ABB RobotStudio station: Arc_Welding.rsstn

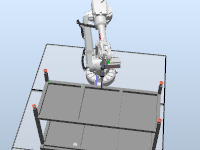
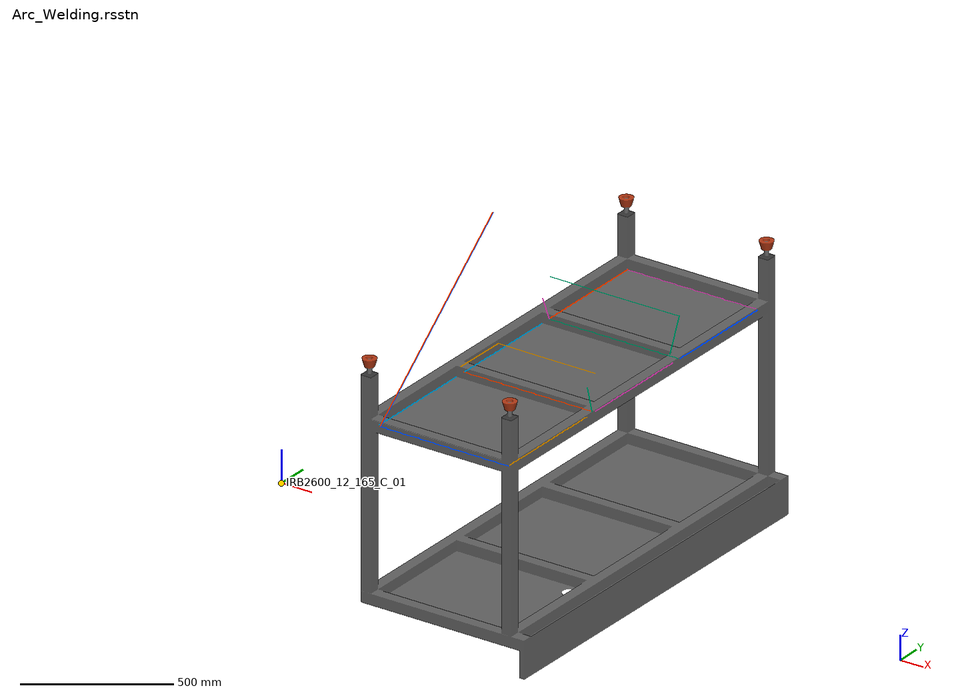
[picture v1: parts stored in the station drawn from their meshes, with robot base, taught points and paths (robot models come from the ABB library and are not in the file)]
Station Arc_Welding (saved by RobotStudio 21.2.9526.0)
Controller Controller_AW
  mechanical unit ROB_1: IRB2600_12_165_C_01, 6 joints, base frame (-416.85, 0, 0) mm
Layout (positions relative to the parent item):
  - IRB2600_12_165_C_01 [mechanism, from Robots\IRB2600_12_165_C_01.rslib] at (-416.85, 0, 0) mm; joint values [0.2384, -0.6663, 0.7884, -0.3764, 0.5482, 0.4666] (rad or m)
  - AW_Gun_PSF_25 [mechanism, from Tools\AW_Gun_PSF_25.rslib] at (157.78, 122.92, 962.92) mm, rotated rx -180 ry 54.2 rz -180 deg
  - Assem1 [graphiccomponentgroup] at (445.82, -642.53, 0) mm, rotated rx 180 ry 0 rz 90 deg
    - Stalas [part] at (21.25, 486.55, -28.09) mm, size 1500 x 650 x 920 mm
    - Part 1 [part] at (22.25, -72.45, -850.09) mm, size 40 x 40 x 35 mm
    - Part 2 [part] at (82.25, -92.45, -879.85) mm, rotated rx 180 ry 0 rz 0 deg, size 51.1 x 51 x 30 mm
    - Hex structural bolt grade C short thread ISO 7412 [part] at (42.25, -92.45, -889.85) mm, rotated rx 180 ry 0 rz 0 deg, size 31.2 x 27 x 80 mm
    - Chamfered plain washer normal ISO 7090 [part] at (42.25, -92.45, -848.59) mm, size 30 x 29.8 x 3 mm
    - Hex flange nut ISO 4161 [part] at (42.25, -92.45, -839.09) mm, size 34.5 x 34.4 x 16 mm
    - Chamfered plain washer normal ISO 7090 [part] at (42.25, 465.55, -848.59) mm, size 30 x 29.8 x 3 mm
    - Hex flange nut ISO 4161 [part] at (42.25, 465.55, -839.09) mm, size 34.5 x 34.4 x 16 mm
    - Hex structural bolt grade C short thread ISO 7412 [part] at (42.25, 465.55, -889.85) mm, rotated rx 180 ry 0 rz 0 deg, size 31.2 x 27 x 80 mm
    - Part 1 [part] at (22.25, 485.55, -850.09) mm, size 40 x 40 x 35 mm
    - Part 2 [part] at (82.25, 465.55, -879.85) mm, rotated rx 180 ry 0 rz 0 deg, size 51.1 x 51 x 30 mm
    - Chamfered plain washer normal ISO 7090 [part] at (1500.25, 465.55, -848.59) mm, size 30 x 29.8 x 3 mm
    - Hex flange nut ISO 4161 [part] at (1500.25, 465.55, -839.09) mm, size 34.5 x 34.4 x 16 mm
    - Hex structural bolt grade C short thread ISO 7412 [part] at (1500.25, 465.55, -889.85) mm, rotated rx 180 ry 0 rz 0 deg, size 31.2 x 27 x 80 mm
    - Part 1 [part] at (1480.25, 485.55, -850.09) mm, size 40 x 40 x 35 mm
    - Part 2 [part] at (1540.25, 465.55, -879.85) mm, rotated rx 180 ry 0 rz 0 deg, size 51.1 x 51 x 30 mm
    - Chamfered plain washer normal ISO 7090 [part] at (1500.25, -92.45, -848.59) mm, size 30 x 29.8 x 3 mm
    - Hex flange nut ISO 4161 [part] at (1500.25, -92.45, -839.09) mm, size 34.5 x 34.4 x 16 mm
    - Hex structural bolt grade C short thread ISO 7412 [part] at (1500.25, -92.45, -889.85) mm, rotated rx 180 ry 0 rz 0 deg, size 31.2 x 27 x 80 mm
    - Part 1 [part] at (1480.25, -72.45, -850.09) mm, size 40 x 40 x 35 mm
    - Part 2 [part] at (1540.25, -92.45, -879.85) mm, rotated rx 180 ry 0 rz 0 deg, size 51.1 x 51 x 30 mm
    - Part 1 [part] at (62.25, 445.55, -28.09) mm, size 1418 x 598 x 40 mm
    - Part 1 [part] at (62.25, 445.55, -660.09) mm, size 1418 x 598 x 40 mm
    - Part 1 [part] at (64.25, 445.55, -660.09) mm, rotated rx 0 ry 90 rz 0 deg, size 40 x 519 x 40 mm
    - Part 1 [part] at (1478.25, 446.55, -660.09) mm, size 40 x 519 x 40 mm
    - Part 1 [part] at (1480.25, 445.55, -28.09) mm, size 40 x 519 x 40 mm
    - Part 1 [part] at (22.25, 445.55, -28.09) mm, size 40 x 519 x 40 mm
Attachment: AW_Gun_PSF_25 is attached to IRB2600_12_165_C_01 / Link6
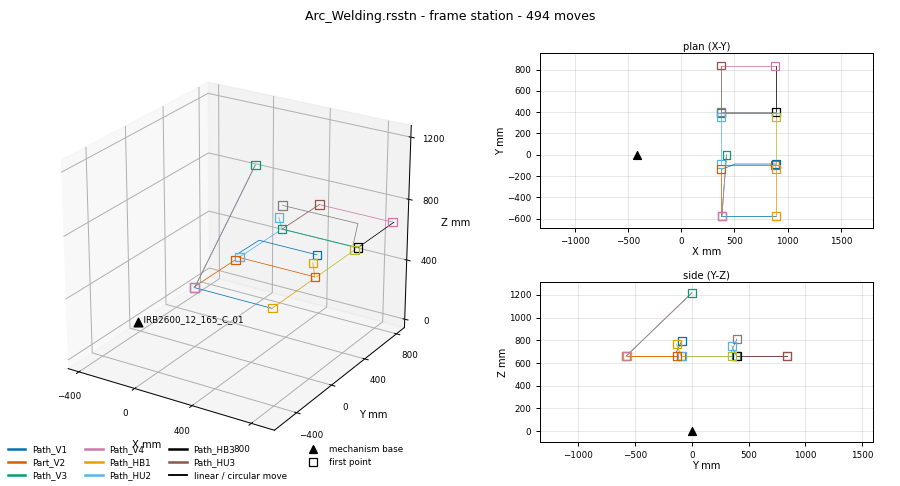
[picture p0: tool path of Arc_Welding.rsstn in frame station, 494 of 494 moves have a stored position in this frame; points joined in program order, loops and branches not executed]
Targets, tools, work objects and paths stored in the station, written as RAPID:
! task T_ROB1
MODULE CalibData
  PERS tooldata AW_Gun:=[TRUE,[[119.5,0,352],[0.890213743,0,0.455543074,0]],[1,[0,0,100],[1,0,0,0],0,0,0]];
ENDMODULE

! task T_ROB1
MODULE Module1
  CONST robtarget Target_10:=[[891.374984158,-578.28436321,660.090342283],[0,0,1,0],[0,0,0,0],[9E+09,9E+09,9E+09,9E+09,9E+09,9E+09]];
  CONST robtarget Target_20:=[[881.374984158,-578.28436321,660.090342283],[0,0,1,0],[0,0,0,0],[9E+09,9E+09,9E+09,9E+09,9E+09,9E+09]];
  CONST robtarget Target_30:=[[871.374984158,-578.28436321,660.090342283],[0,0,1,0],[0,0,0,0],[9E+09,9E+09,9E+09,9E+09,9E+09,9E+09]];
  CONST robtarget Target_40:=[[861.374984158,-578.28436321,660.090342283],[0,0,1,0],[0,0,0,0],[9E+09,9E+09,9E+09,9E+09,9E+09,9E+09]];
  CONST robtarget Target_50:=[[851.374984158,-578.28436321,660.090342283],[0,0,1,0],[0,0,0,0],[9E+09,9E+09,9E+09,9E+09,9E+09,9E+09]];
  CONST robtarget Target_60:=[[841.374984158,-578.28436321,660.090342283],[0,0,1,0],[0,0,0,0],[9E+09,9E+09,9E+09,9E+09,9E+09,9E+09]];
  CONST robtarget Target_70:=[[831.374984158,-578.28436321,660.090342283],[0,0,1,0],[0,0,0,0],[9E+09,9E+09,9E+09,9E+09,9E+09,9E+09]];
  CONST robtarget Target_80:=[[821.374984158,-578.28436321,660.090342283],[0,0,1,0],[0,0,0,0],[9E+09,9E+09,9E+09,9E+09,9E+09,9E+09]];
  CONST robtarget Target_90:=[[811.374984158,-578.28436321,660.090342283],[0,0,1,0],[0,0,0,0],[9E+09,9E+09,9E+09,9E+09,9E+09,9E+09]];
  CONST robtarget Target_100:=[[801.374984158,-578.28436321,660.090342283],[0,0,1,0],[0,0,0,0],[9E+09,9E+09,9E+09,9E+09,9E+09,9E+09]];
  CONST robtarget Target_110:=[[791.374984158,-578.28436321,660.090342283],[0,0,1,0],[0,0,0,0],[9E+09,9E+09,9E+09,9E+09,9E+09,9E+09]];
  CONST robtarget Target_120:=[[781.374984158,-578.28436321,660.090342283],[0,0,1,0],[0,0,0,0],[9E+09,9E+09,9E+09,9E+09,9E+09,9E+09]];
  CONST robtarget Target_130:=[[771.374984158,-578.28436321,660.090342283],[0,0,1,0],[0,0,0,0],[9E+09,9E+09,9E+09,9E+09,9E+09,9E+09]];
  CONST robtarget Target_140:=[[761.374984158,-578.28436321,660.090342283],[0,0,1,0],[0,0,0,0],[9E+09,9E+09,9E+09,9E+09,9E+09,9E+09]];
  CONST robtarget Target_150:=[[751.374984158,-578.28436321,660.090342283],[0,0,1,0],[0,0,0,0],[9E+09,9E+09,9E+09,9E+09,9E+09,9E+09]];
  CONST robtarget Target_160:=[[741.374984158,-578.28436321,660.090342283],[0,0,1,0],[0,0,0,0],[9E+09,9E+09,9E+09,9E+09,9E+09,9E+09]];
  CONST robtarget Target_170:=[[731.374984158,-578.28436321,660.090342283],[0,0,1,0],[0,0,0,0],[9E+09,9E+09,9E+09,9E+09,9E+09,9E+09]];
  CONST robtarget Target_180:=[[721.374984158,-578.28436321,660.090342283],[0,0,1,0],[0,0,0,0],[9E+09,9E+09,9E+09,9E+09,9E+09,9E+09]];
  CONST robtarget Target_190:=[[711.374984158,-578.28436321,660.090342283],[0,0,1,0],[0,0,0,0],[9E+09,9E+09,9E+09,9E+09,9E+09,9E+09]];
  CONST robtarget Target_200:=[[701.374984158,-578.28436321,660.090342283],[0,0,1,0],[0,0,0,0],[9E+09,9E+09,9E+09,9E+09,9E+09,9E+09]];
  CONST robtarget Target_210:=[[691.374984158,-578.28436321,660.090342283],[0,0,1,0],[0,0,0,0],[9E+09,9E+09,9E+09,9E+09,9E+09,9E+09]];
  CONST robtarget Target_220:=[[681.374984158,-578.28436321,660.090342283],[0,0,1,0],[0,0,0,0],[9E+09,9E+09,9E+09,9E+09,9E+09,9E+09]];
  CONST robtarget Target_230:=[[671.374984158,-578.28436321,660.090342283],[0,0,1,0],[0,0,0,0],[9E+09,9E+09,9E+09,9E+09,9E+09,9E+09]];
  CONST robtarget Target_240:=[[661.374984158,-578.28436321,660.090342283],[0,0,1,0],[0,0,0,0],[9E+09,9E+09,9E+09,9E+09,9E+09,9E+09]];
  CONST robtarget Target_250:=[[651.374984158,-578.28436321,660.090342283],[0,0,1,0],[0,0,0,0],[9E+09,9E+09,9E+09,9E+09,9E+09,9E+09]];
  CONST robtarget Target_260:=[[641.374984158,-578.28436321,660.090342283],[0,0,1,0],[0,0,0,0],[9E+09,9E+09,9E+09,9E+09,9E+09,9E+09]];
  CONST robtarget Target_270:=[[631.374984158,-578.28436321,660.090342283],[0,0,1,0],[0,0,0,0],[9E+09,9E+09,9E+09,9E+09,9E+09,9E+09]];
  CONST robtarget Target_280:=[[621.374984158,-578.28436321,660.090342283],[0,0,1,0],[0,0,0,0],[9E+09,9E+09,9E+09,9E+09,9E+09,9E+09]];
  CONST robtarget Target_290:=[[611.374984158,-578.28436321,660.090342283],[0,0,1,0],[0,0,0,0],[9E+09,9E+09,9E+09,9E+09,9E+09,9E+09]];
  CONST robtarget Target_300:=[[601.374984158,-578.28436321,660.090342283],[0,0,1,0],[0,0,0,0],[9E+09,9E+09,9E+09,9E+09,9E+09,9E+09]];
  CONST robtarget Target_310:=[[591.374984158,-578.28436321,660.090342283],[0,0,1,0],[0,0,0,0],[9E+09,9E+09,9E+09,9E+09,9E+09,9E+09]];
  CONST robtarget Target_320:=[[581.374984158,-578.28436321,660.090342283],[0,0,1,0],[0,0,0,0],[9E+09,9E+09,9E+09,9E+09,9E+09,9E+09]];
  CONST robtarget Target_330:=[[571.374984158,-578.28436321,660.090342283],[0,0,1,0],[0,0,0,0],[9E+09,9E+09,9E+09,9E+09,9E+09,9E+09]];
  CONST robtarget Target_340:=[[561.374984158,-578.28436321,660.090342283],[0,0,1,0],[0,0,0,0],[9E+09,9E+09,9E+09,9E+09,9E+09,9E+09]];
  CONST robtarget Target_350:=[[551.374984158,-578.28436321,660.090342283],[0,0,1,0],[0,0,0,0],[9E+09,9E+09,9E+09,9E+09,9E+09,9E+09]];
  CONST robtarget Target_360:=[[541.374984158,-578.28436321,660.090342283],[0,0,1,0],[0,0,0,0],[9E+09,9E+09,9E+09,9E+09,9E+09,9E+09]];
  CONST robtarget Target_370:=[[531.374984158,-578.28436321,660.090342283],[0,0,1,0],[0,0,0,0],[9E+09,9E+09,9E+09,9E+09,9E+09,9E+09]];
  CONST robtarget Target_380:=[[521.374984158,-578.28436321,660.090342283],[0,0,1,0],[0,0,0,0],[9E+09,9E+09,9E+09,9E+09,9E+09,9E+09]];
  CONST robtarget Target_390:=[[511.374984158,-578.28436321,660.090342283],[0,0,1,0],[0,0,0,0],[9E+09,9E+09,9E+09,9E+09,9E+09,9E+09]];
  CONST robtarget Target_400:=[[501.374984158,-578.28436321,660.090342283],[0,0,1,0],[0,0,0,0],[9E+09,9E+09,9E+09,9E+09,9E+09,9E+09]];
  CONST robtarget Target_410:=[[491.374984158,-578.28436321,660.090342283],[0,0,1,0],[0,0,0,0],[9E+09,9E+09,9E+09,9E+09,9E+09,9E+09]];
  CONST robtarget Target_420:=[[481.374984158,-578.28436321,660.090342283],[0,0,1,0],[0,0,0,0],[9E+09,9E+09,9E+09,9E+09,9E+09,9E+09]];
  CONST robtarget Target_430:=[[471.374984158,-578.28436321,660.090342283],[0,0,1,0],[0,0,0,0],[9E+09,9E+09,9E+09,9E+09,9E+09,9E+09]];
  CONST robtarget Target_440:=[[461.374984158,-578.28436321,660.090342283],[0,0,1,0],[0,0,0,0],[9E+09,9E+09,9E+09,9E+09,9E+09,9E+09]];
  CONST robtarget Target_450:=[[451.374984158,-578.28436321,660.090342283],[0,0,1,0],[0,0,0,0],[9E+09,9E+09,9E+09,9E+09,9E+09,9E+09]];
  CONST robtarget Target_460:=[[441.374984158,-578.28436321,660.090342283],[0,0,1,0],[0,0,0,0],[9E+09,9E+09,9E+09,9E+09,9E+09,9E+09]];
  CONST robtarget Target_470:=[[431.374984158,-578.28436321,660.090342283],[0,0,1,0],[0,0,0,0],[9E+09,9E+09,9E+09,9E+09,9E+09,9E+09]];
  CONST robtarget Target_480:=[[421.374984158,-578.28436321,660.090342283],[0,0,1,0],[0,0,0,0],[9E+09,9E+09,9E+09,9E+09,9E+09,9E+09]];
  CONST robtarget Target_490:=[[411.374984158,-578.28436321,660.090342283],[0,0,1,0],[0,0,0,0],[9E+09,9E+09,9E+09,9E+09,9E+09,9E+09]];
  CONST robtarget Target_500:=[[401.374984158,-578.28436321,660.090342283],[0,0,1,0],[0,0,0,0],[9E+09,9E+09,9E+09,9E+09,9E+09,9E+09]];
  CONST robtarget Target_510:=[[391.374984158,-578.28436321,660.090342283],[0,0,1,0],[0,0,0,0],[9E+09,9E+09,9E+09,9E+09,9E+09,9E+09]];
  CONST robtarget Target_520:=[[381.374984158,-578.28436321,660.090342283],[0,0,1,0],[0,0,0,0],[9E+09,9E+09,9E+09,9E+09,9E+09,9E+09]];
  CONST robtarget Target_530:=[[373.374984158,-133.68436321,660.090342283],[0.5,0.5,-0.5,-0.5],[0,0,0,0],[9E+09,9E+09,9E+09,9E+09,9E+09,9E+09]];
  CONST robtarget Target_540:=[[373.374984158,-580.28436321,660.090342283],[0.5,0.5,-0.5,-0.5],[0,0,0,0],[9E+09,9E+09,9E+09,9E+09,9E+09,9E+09]];
  CONST robtarget Target_570:=[[373.374984158,-93.68436321,660.090342283],[0,0,1,0],[0,0,0,0],[9E+09,9E+09,9E+09,9E+09,9E+09,9E+09]];
  CONST robtarget Target_580:=[[383.374984158,-93.68436321,660.090342283],[0,0,1,0],[0,0,0,0],[9E+09,9E+09,9E+09,9E+09,9E+09,9E+09]];
  CONST robtarget Target_590:=[[393.374984158,-93.68436321,660.090342283],[0,0,1,0],[0,0,0,0],[9E+09,9E+09,9E+09,9E+09,9E+09,9E+09]];
  CONST robtarget Target_600:=[[403.374984158,-93.68436321,660.090342283],[0,0,1,0],[0,0,0,0],[9E+09,9E+09,9E+09,9E+09,9E+09,9E+09]];
  CONST robtarget Target_610:=[[413.374984158,-93.68436321,660.090342283],[0,0,1,0],[0,0,0,0],[9E+09,9E+09,9E+09,9E+09,9E+09,9E+09]];
  CONST robtarget Target_620:=[[423.374984158,-93.68436321,660.090342283],[0,0,1,0],[0,0,0,0],[9E+09,9E+09,9E+09,9E+09,9E+09,9E+09]];
  CONST robtarget Target_630:=[[433.374984158,-93.68436321,660.090342283],[0,0,1,0],[0,0,0,0],[9E+09,9E+09,9E+09,9E+09,9E+09,9E+09]];
  CONST robtarget Target_640:=[[443.374984158,-93.68436321,660.090342283],[0,0,1,0],[0,0,0,0],[9E+09,9E+09,9E+09,9E+09,9E+09,9E+09]];
  CONST robtarget Target_650:=[[453.374984158,-93.68436321,660.090342283],[0,0,1,0],[0,0,0,0],[9E+09,9E+09,9E+09,9E+09,9E+09,9E+09]];
  CONST robtarget Target_660:=[[463.374984158,-93.68436321,660.090342283],[0,0,1,0],[0,0,0,0],[9E+09,9E+09,9E+09,9E+09,9E+09,9E+09]];
  CONST robtarget Target_670:=[[473.374984158,-93.68436321,660.090342283],[0,0,1,0],[0,0,0,0],[9E+09,9E+09,9E+09,9E+09,9E+09,9E+09]];
  CONST robtarget Target_680:=[[483.374984158,-93.68436321,660.090342283],[0,0,1,0],[0,0,0,0],[9E+09,9E+09,9E+09,9E+09,9E+09,9E+09]];
  CONST robtarget Target_690:=[[493.374984158,-93.68436321,660.090342283],[0,0,1,0],[0,0,0,0],[9E+09,9E+09,9E+09,9E+09,9E+09,9E+09]];
  CONST robtarget Target_700:=[[503.374984158,-93.68436321,660.090342283],[0,0,1,0],[0,0,0,0],[9E+09,9E+09,9E+09,9E+09,9E+09,9E+09]];
  CONST robtarget Target_710:=[[513.374984158,-93.68436321,660.090342283],[0,0,1,0],[0,0,0,0],[9E+09,9E+09,9E+09,9E+09,9E+09,9E+09]];
  CONST robtarget Target_720:=[[523.374984158,-93.68436321,660.090342283],[0,0,1,0],[0,0,0,0],[9E+09,9E+09,9E+09,9E+09,9E+09,9E+09]];
  CONST robtarget Target_730:=[[533.374984158,-93.68436321,660.090342283],[0,0,1,0],[0,0,0,0],[9E+09,9E+09,9E+09,9E+09,9E+09,9E+09]];
  CONST robtarget Target_740:=[[543.374984158,-93.68436321,660.090342283],[0,0,1,0],[0,0,0,0],[9E+09,9E+09,9E+09,9E+09,9E+09,9E+09]];
  CONST robtarget Target_750:=[[553.374984158,-93.68436321,660.090342283],[0,0,1,0],[0,0,0,0],[9E+09,9E+09,9E+09,9E+09,9E+09,9E+09]];
  CONST robtarget Target_760:=[[563.374984158,-93.68436321,660.090342283],[0,0,1,0],[0,0,0,0],[9E+09,9E+09,9E+09,9E+09,9E+09,9E+09]];
  CONST robtarget Target_770:=[[573.374984158,-93.68436321,660.090342283],[0,0,1,0],[0,0,0,0],[9E+09,9E+09,9E+09,9E+09,9E+09,9E+09]];
  CONST robtarget Target_780:=[[583.374984158,-93.68436321,660.090342283],[0,0,1,0],[0,0,0,0],[9E+09,9E+09,9E+09,9E+09,9E+09,9E+09]];
  CONST robtarget Target_790:=[[593.374984158,-93.68436321,660.090342283],[0,0,1,0],[0,0,0,0],[9E+09,9E+09,9E+09,9E+09,9E+09,9E+09]];
  CONST robtarget Target_800:=[[603.374984158,-93.68436321,660.090342283],[0,0,1,0],[0,0,0,0],[9E+09,9E+09,9E+09,9E+09,9E+09,9E+09]];
  CONST robtarget Target_810:=[[613.374984158,-93.68436321,660.090342283],[0,0,1,0],[0,0,0,0],[9E+09,9E+09,9E+09,9E+09,9E+09,9E+09]];
  CONST robtarget Target_820:=[[623.374984158,-93.68436321,660.090342283],[0,0,1,0],[0,0,0,0],[9E+09,9E+09,9E+09,9E+09,9E+09,9E+09]];
  CONST robtarget Target_830:=[[633.374984158,-93.68436321,660.090342283],[0,0,1,0],[0,0,0,0],[9E+09,9E+09,9E+09,9E+09,9E+09,9E+09]];
  CONST robtarget Target_840:=[[643.374984158,-93.68436321,660.090342283],[0,0,1,0],[0,0,0,0],[9E+09,9E+09,9E+09,9E+09,9E+09,9E+09]];
  CONST robtarget Target_850:=[[653.374984158,-93.68436321,660.090342283],[0,0,1,0],[0,0,0,0],[9E+09,9E+09,9E+09,9E+09,9E+09,9E+09]];
  CONST robtarget Target_860:=[[663.374984158,-93.68436321,660.090342283],[0,0,1,0],[0,0,0,0],[9E+09,9E+09,9E+09,9E+09,9E+09,9E+09]];
  CONST robtarget Target_870:=[[673.374984158,-93.68436321,660.090342283],[0,0,1,0],[0,0,0,0],[9E+09,9E+09,9E+09,9E+09,9E+09,9E+09]];
  CONST robtarget Target_880:=[[683.374984158,-93.68436321,660.090342283],[0,0,1,0],[0,0,0,0],[9E+09,9E+09,9E+09,9E+09,9E+09,9E+09]];
  CONST robtarget Target_890:=[[693.374984158,-93.68436321,660.090342283],[0,0,1,0],[0,0,0,0],[9E+09,9E+09,9E+09,9E+09,9E+09,9E+09]];
  CONST robtarget Target_900:=[[703.374984158,-93.68436321,660.090342283],[0,0,1,0],[0,0,0,0],[9E+09,9E+09,9E+09,9E+09,9E+09,9E+09]];
  CONST robtarget Target_910:=[[713.374984158,-93.68436321,660.090342283],[0,0,1,0],[0,0,0,0],[9E+09,9E+09,9E+09,9E+09,9E+09,9E+09]];
  CONST robtarget Target_920:=[[723.374984158,-93.68436321,660.090342283],[0,0,1,0],[0,0,0,0],[9E+09,9E+09,9E+09,9E+09,9E+09,9E+09]];
  CONST robtarget Target_930:=[[733.374984158,-93.68436321,660.090342283],[0,0,1,0],[0,0,0,0],[9E+09,9E+09,9E+09,9E+09,9E+09,9E+09]];
  CONST robtarget Target_940:=[[743.374984158,-93.68436321,660.090342283],[0,0,1,0],[0,0,0,0],[9E+09,9E+09,9E+09,9E+09,9E+09,9E+09]];
  CONST robtarget Target_950:=[[753.374984158,-93.68436321,660.090342283],[0,0,1,0],[0,0,0,0],[9E+09,9E+09,9E+09,9E+09,9E+09,9E+09]];
  CONST robtarget Target_960:=[[763.374984158,-93.68436321,660.090342283],[0,0,1,0],[0,0,0,0],[9E+09,9E+09,9E+09,9E+09,9E+09,9E+09]];
  CONST robtarget Target_970:=[[773.374984158,-93.68436321,660.090342283],[0,0,1,0],[0,0,0,0],[9E+09,9E+09,9E+09,9E+09,9E+09,9E+09]];
  CONST robtarget Target_980:=[[783.374984158,-93.68436321,660.090342283],[0,0,1,0],[0,0,0,0],[9E+09,9E+09,9E+09,9E+09,9E+09,9E+09]];
  CONST robtarget Target_990:=[[793.374984158,-93.68436321,660.090342283],[0,0,1,0],[0,0,0,0],[9E+09,9E+09,9E+09,9E+09,9E+09,9E+09]];
  CONST robtarget Target_1000:=[[803.374984158,-93.68436321,660.090342283],[0,0,1,0],[0,0,0,0],[9E+09,9E+09,9E+09,9E+09,9E+09,9E+09]];
  CONST robtarget Target_1010:=[[813.374984158,-93.68436321,660.090342283],[0,0,1,0],[0,0,0,0],[9E+09,9E+09,9E+09,9E+09,9E+09,9E+09]];
  CONST robtarget Target_1020:=[[823.374984158,-93.68436321,660.090342283],[0,0,1,0],[0,0,0,0],[9E+09,9E+09,9E+09,9E+09,9E+09,9E+09]];
  CONST robtarget Target_1030:=[[833.374984158,-93.68436321,660.090342283],[0,0,1,0],[0,0,0,0],[9E+09,9E+09,9E+09,9E+09,9E+09,9E+09]];
  CONST robtarget Target_1040:=[[843.374984158,-93.68436321,660.090342283],[0,0,1,0],[0,0,0,0],[9E+09,9E+09,9E+09,9E+09,9E+09,9E+09]];
  CONST robtarget Target_1050:=[[853.374984158,-93.68436321,660.090342283],[0,0,1,0],[0,0,0,0],[9E+09,9E+09,9E+09,9E+09,9E+09,9E+09]];
  CONST robtarget Target_1060:=[[863.374984158,-93.68436321,660.090342283],[0,0,1,0],[0,0,0,0],[9E+09,9E+09,9E+09,9E+09,9E+09,9E+09]];
  CONST robtarget Target_1070:=[[873.374984158,-93.68436321,660.090342283],[0,0,1,0],[0,0,0,0],[9E+09,9E+09,9E+09,9E+09,9E+09,9E+09]];
  CONST robtarget Target_1080:=[[883.374984158,-93.68436321,660.090342283],[0,0,1,0],[0,0,0,0],[9E+09,9E+09,9E+09,9E+09,9E+09,9E+09]];
  CONST robtarget Target_1090:=[[373.374984158,392.91563679,660.090342283],[0,0,1,0],[0,0,0,0],[9E+09,9E+09,9E+09,9E+09,9E+09,9E+09]];
  CONST robtarget Target_1100:=[[383.374984158,392.91563679,660.090342283],[0,0,1,0],[0,0,0,0],[9E+09,9E+09,9E+09,9E+09,9E+09,9E+09]];
  CONST robtarget Target_1110:=[[393.374984158,392.91563679,660.090342283],[0,0,1,0],[0,0,0,0],[9E+09,9E+09,9E+09,9E+09,9E+09,9E+09]];
  CONST robtarget Target_1120:=[[403.374984158,392.91563679,660.090342283],[0,0,1,0],[0,0,0,0],[9E+09,9E+09,9E+09,9E+09,9E+09,9E+09]];
  CONST robtarget Target_1130:=[[413.374984158,392.91563679,660.090342283],[0,0,1,0],[0,0,0,0],[9E+09,9E+09,9E+09,9E+09,9E+09,9E+09]];
  CONST robtarget Target_1140:=[[423.374984158,392.91563679,660.090342283],[0,0,1,0],[0,0,0,0],[9E+09,9E+09,9E+09,9E+09,9E+09,9E+09]];
  CONST robtarget Target_1150:=[[433.374984158,392.91563679,660.090342283],[0,0,1,0],[0,0,0,0],[9E+09,9E+09,9E+09,9E+09,9E+09,9E+09]];
  CONST robtarget Target_1160:=[[443.374984158,392.91563679,660.090342283],[0,0,1,0],[0,0,0,0],[9E+09,9E+09,9E+09,9E+09,9E+09,9E+09]];
  CONST robtarget Target_1170:=[[453.374984158,392.91563679,660.090342283],[0,0,1,0],[0,0,0,0],[9E+09,9E+09,9E+09,9E+09,9E+09,9E+09]];
  CONST robtarget Target_1180:=[[463.374984158,392.91563679,660.090342283],[0,0,1,0],[0,0,0,0],[9E+09,9E+09,9E+09,9E+09,9E+09,9E+09]];
  CONST robtarget Target_1190:=[[473.374984158,392.91563679,660.090342283],[0,0,1,0],[0,0,0,0],[9E+09,9E+09,9E+09,9E+09,9E+09,9E+09]];
  CONST robtarget Target_1200:=[[483.374984158,392.91563679,660.090342283],[0,0,1,0],[0,0,0,0],[9E+09,9E+09,9E+09,9E+09,9E+09,9E+09]];
  CONST robtarget Target_1210:=[[493.374984158,392.91563679,660.090342283],[0,0,1,0],[0,0,0,0],[9E+09,9E+09,9E+09,9E+09,9E+09,9E+09]];
  CONST robtarget Target_1220:=[[503.374984158,392.91563679,660.090342283],[0,0,1,0],[0,0,0,0],[9E+09,9E+09,9E+09,9E+09,9E+09,9E+09]];
  CONST robtarget Target_1230:=[[513.374984158,392.91563679,660.090342283],[0,0,1,0],[0,0,0,0],[9E+09,9E+09,9E+09,9E+09,9E+09,9E+09]];
  CONST robtarget Target_1240:=[[523.374984158,392.91563679,660.090342283],[0,0,1,0],[0,0,0,0],[9E+09,9E+09,9E+09,9E+09,9E+09,9E+09]];
  CONST robtarget Target_1250:=[[533.374984158,392.91563679,660.090342283],[0,0,1,0],[0,0,0,0],[9E+09,9E+09,9E+09,9E+09,9E+09,9E+09]];
  CONST robtarget Target_1260:=[[543.374984158,392.91563679,660.090342283],[0,0,1,0],[0,0,0,0],[9E+09,9E+09,9E+09,9E+09,9E+09,9E+09]];
  CONST robtarget Target_1270:=[[553.374984158,392.91563679,660.090342283],[0,0,1,0],[0,0,0,0],[9E+09,9E+09,9E+09,9E+09,9E+09,9E+09]];
  CONST robtarget Target_1280:=[[563.374984158,392.91563679,660.090342283],[0,0,1,0],[0,0,0,0],[9E+09,9E+09,9E+09,9E+09,9E+09,9E+09]];
  CONST robtarget Target_1290:=[[573.374984158,392.91563679,660.090342283],[0,0,1,0],[0,0,0,0],[9E+09,9E+09,9E+09,9E+09,9E+09,9E+09]];
  CONST robtarget Target_1300:=[[583.374984158,392.91563679,660.090342283],[0,0,1,0],[0,0,0,0],[9E+09,9E+09,9E+09,9E+09,9E+09,9E+09]];
  CONST robtarget Target_1310:=[[593.374984158,392.91563679,660.090342283],[0,0,1,0],[0,0,0,0],[9E+09,9E+09,9E+09,9E+09,9E+09,9E+09]];
  CONST robtarget Target_1320:=[[603.374984158,392.91563679,660.090342283],[0,0,1,0],[0,0,0,0],[9E+09,9E+09,9E+09,9E+09,9E+09,9E+09]];
  CONST robtarget Target_1330:=[[613.374984158,392.91563679,660.090342283],[0,0,1,0],[0,0,0,0],[9E+09,9E+09,9E+09,9E+09,9E+09,9E+09]];
  CONST robtarget Target_1340:=[[623.374984158,392.91563679,660.090342283],[0,0,1,0],[0,0,0,0],[9E+09,9E+09,9E+09,9E+09,9E+09,9E+09]];
  CONST robtarget Target_1350:=[[633.374984158,392.91563679,660.090342283],[0,0,1,0],[0,0,0,0],[9E+09,9E+09,9E+09,9E+09,9E+09,9E+09]];
  CONST robtarget Target_1360:=[[643.374984158,392.91563679,660.090342283],[0,0,1,0],[0,0,0,0],[9E+09,9E+09,9E+09,9E+09,9E+09,9E+09]];
  CONST robtarget Target_1370:=[[653.374984158,392.91563679,660.090342283],[0,0,1,0],[0,0,0,0],[9E+09,9E+09,9E+09,9E+09,9E+09,9E+09]];
  CONST robtarget Target_1380:=[[663.374984158,392.91563679,660.090342283],[0,0,1,0],[0,0,0,0],[9E+09,9E+09,9E+09,9E+09,9E+09,9E+09]];
  CONST robtarget Target_1390:=[[673.374984158,392.91563679,660.090342283],[0,0,1,0],[0,0,0,0],[9E+09,9E+09,9E+09,9E+09,9E+09,9E+09]];
  CONST robtarget Target_1400:=[[683.374984158,392.91563679,660.090342283],[0,0,1,0],[0,0,0,0],[9E+09,9E+09,9E+09,9E+09,9E+09,9E+09]];
  CONST robtarget Target_1410:=[[693.374984158,392.91563679,660.090342283],[0,0,1,0],[0,0,0,0],[9E+09,9E+09,9E+09,9E+09,9E+09,9E+09]];
  CONST robtarget Target_1420:=[[703.374984158,392.91563679,660.090342283],[0,0,1,0],[0,0,0,0],[9E+09,9E+09,9E+09,9E+09,9E+09,9E+09]];
  CONST robtarget Target_1430:=[[713.374984158,392.91563679,660.090342283],[0,0,1,0],[0,0,0,0],[9E+09,9E+09,9E+09,9E+09,9E+09,9E+09]];
  CONST robtarget Target_1440:=[[723.374984158,392.91563679,660.090342283],[0,0,1,0],[0,0,0,0],[9E+09,9E+09,9E+09,9E+09,9E+09,9E+09]];
  CONST robtarget Target_1450:=[[733.374984158,392.91563679,660.090342283],[0,0,1,0],[0,0,0,0],[9E+09,9E+09,9E+09,9E+09,9E+09,9E+09]];
  CONST robtarget Target_1460:=[[743.374984158,392.91563679,660.090342283],[0,0,1,0],[0,0,0,0],[9E+09,9E+09,9E+09,9E+09,9E+09,9E+09]];
  CONST robtarget Target_1470:=[[753.374984158,392.91563679,660.090342283],[0,0,1,0],[0,0,0,0],[9E+09,9E+09,9E+09,9E+09,9E+09,9E+09]];
  CONST robtarget Target_1480:=[[763.374984158,392.91563679,660.090342283],[0,0,1,0],[0,0,0,0],[9E+09,9E+09,9E+09,9E+09,9E+09,9E+09]];
  CONST robtarget Target_1490:=[[773.374984158,392.91563679,660.090342283],[0,0,1,0],[0,0,0,0],[9E+09,9E+09,9E+09,9E+09,9E+09,9E+09]];
  CONST robtarget Target_1500:=[[783.374984158,392.91563679,660.090342283],[0,0,1,0],[0,0,0,0],[9E+09,9E+09,9E+09,9E+09,9E+09,9E+09]];
  CONST robtarget Target_1510:=[[793.374984158,392.91563679,660.090342283],[0,0,1,0],[0,0,0,0],[9E+09,9E+09,9E+09,9E+09,9E+09,9E+09]];
  CONST robtarget Target_1520:=[[803.374984158,392.91563679,660.090342283],[0,0,1,0],[0,0,0,0],[9E+09,9E+09,9E+09,9E+09,9E+09,9E+09]];
  CONST robtarget Target_1530:=[[813.374984158,392.91563679,660.090342283],[0,0,1,0],[0,0,0,0],[9E+09,9E+09,9E+09,9E+09,9E+09,9E+09]];
  CONST robtarget Target_1540:=[[823.374984158,392.91563679,660.090342283],[0,0,1,0],[0,0,0,0],[9E+09,9E+09,9E+09,9E+09,9E+09,9E+09]];
  CONST robtarget Target_1550:=[[833.374984158,392.91563679,660.090342283],[0,0,1,0],[0,0,0,0],[9E+09,9E+09,9E+09,9E+09,9E+09,9E+09]];
  CONST robtarget Target_1560:=[[843.374984158,392.91563679,660.090342283],[0,0,1,0],[0,0,0,0],[9E+09,9E+09,9E+09,9E+09,9E+09,9E+09]];
  CONST robtarget Target_1570:=[[853.374984158,392.91563679,660.090342283],[0,0,1,0],[0,0,0,0],[9E+09,9E+09,9E+09,9E+09,9E+09,9E+09]];
  CONST robtarget Target_1580:=[[863.374984158,392.91563679,660.090342283],[0,0,1,0],[0,0,0,0],[9E+09,9E+09,9E+09,9E+09,9E+09,9E+09]];
  CONST robtarget Target_1590:=[[873.374984158,392.91563679,660.090342283],[0,0,1,0],[0,0,0,0],[9E+09,9E+09,9E+09,9E+09,9E+09,9E+09]];
  CONST robtarget Target_1600:=[[883.374984158,392.91563679,660.090342283],[0,0,1,0],[0,0,0,0],[9E+09,9E+09,9E+09,9E+09,9E+09,9E+09]];
  CONST robtarget Target_1610:=[[373.374984158,835.71563679,660.090342283],[0,0,1,0],[0,0,0,0],[9E+09,9E+09,9E+09,9E+09,9E+09,9E+09]];
  CONST robtarget Target_1620:=[[383.374984158,835.71563679,660.090342283],[0,0,1,0],[0,0,0,0],[9E+09,9E+09,9E+09,9E+09,9E+09,9E+09]];
  CONST robtarget Target_1630:=[[393.374984158,835.71563679,660.090342283],[0,0,1,0],[0,0,0,0],[9E+09,9E+09,9E+09,9E+09,9E+09,9E+09]];
  CONST robtarget Target_1640:=[[403.374984158,835.71563679,660.090342283],[0,0,1,0],[0,0,0,0],[9E+09,9E+09,9E+09,9E+09,9E+09,9E+09]];
  CONST robtarget Target_1650:=[[413.374984158,835.71563679,660.090342283],[0,0,1,0],[0,0,0,0],[9E+09,9E+09,9E+09,9E+09,9E+09,9E+09]];
  CONST robtarget Target_1660:=[[423.374984158,835.71563679,660.090342283],[0,0,1,0],[0,0,0,0],[9E+09,9E+09,9E+09,9E+09,9E+09,9E+09]];
  CONST robtarget Target_1670:=[[433.374984158,835.71563679,660.090342283],[0,0,1,0],[0,0,0,0],[9E+09,9E+09,9E+09,9E+09,9E+09,9E+09]];
  CONST robtarget Target_1680:=[[443.374984158,835.71563679,660.090342283],[0,0,1,0],[0,0,0,0],[9E+09,9E+09,9E+09,9E+09,9E+09,9E+09]];
  CONST robtarget Target_1690:=[[453.374984158,835.71563679,660.090342283],[0,0,1,0],[0,0,0,0],[9E+09,9E+09,9E+09,9E+09,9E+09,9E+09]];
  CONST robtarget Target_1700:=[[463.374984158,835.71563679,660.090342283],[0,0,1,0],[0,0,0,0],[9E+09,9E+09,9E+09,9E+09,9E+09,9E+09]];
  CONST robtarget Target_1710:=[[473.374984158,835.71563679,660.090342283],[0,0,1,0],[0,0,0,0],[9E+09,9E+09,9E+09,9E+09,9E+09,9E+09]];
  CONST robtarget Target_1720:=[[483.374984158,835.71563679,660.090342283],[0,0,1,0],[0,0,0,0],[9E+09,9E+09,9E+09,9E+09,9E+09,9E+09]];
  CONST robtarget Target_1730:=[[493.374984158,835.71563679,660.090342283],[0,0,1,0],[0,0,0,0],[9E+09,9E+09,9E+09,9E+09,9E+09,9E+09]];
  CONST robtarget Target_1740:=[[503.374984158,835.71563679,660.090342283],[0,0,1,0],[0,0,0,0],[9E+09,9E+09,9E+09,9E+09,9E+09,9E+09]];
  CONST robtarget Target_1750:=[[513.374984158,835.71563679,660.090342283],[0,0,1,0],[0,0,0,0],[9E+09,9E+09,9E+09,9E+09,9E+09,9E+09]];
  CONST robtarget Target_1760:=[[523.374984158,835.71563679,660.090342283],[0,0,1,0],[0,0,0,0],[9E+09,9E+09,9E+09,9E+09,9E+09,9E+09]];
  CONST robtarget Target_1770:=[[533.374984158,835.71563679,660.090342283],[0,0,1,0],[0,0,0,0],[9E+09,9E+09,9E+09,9E+09,9E+09,9E+09]];
  CONST robtarget Target_1780:=[[543.374984158,835.71563679,660.090342283],[0,0,1,0],[0,0,0,0],[9E+09,9E+09,9E+09,9E+09,9E+09,9E+09]];
  CONST robtarget Target_1790:=[[553.374984158,835.71563679,660.090342283],[0,0,1,0],[0,0,0,0],[9E+09,9E+09,9E+09,9E+09,9E+09,9E+09]];
  CONST robtarget Target_1800:=[[563.374984158,835.71563679,660.090342283],[0,0,1,0],[0,0,0,0],[9E+09,9E+09,9E+09,9E+09,9E+09,9E+09]];
  CONST robtarget Target_1810:=[[573.374984158,835.71563679,660.090342283],[0,0,1,0],[0,0,0,0],[9E+09,9E+09,9E+09,9E+09,9E+09,9E+09]];
  CONST robtarget Target_1820:=[[583.374984158,835.71563679,660.090342283],[0,0,1,0],[0,0,0,0],[9E+09,9E+09,9E+09,9E+09,9E+09,9E+09]];
  CONST robtarget Target_1830:=[[593.374984158,835.71563679,660.090342283],[0,0,1,0],[0,0,0,0],[9E+09,9E+09,9E+09,9E+09,9E+09,9E+09]];
  CONST robtarget Target_1840:=[[603.374984158,835.71563679,660.090342283],[0,0,1,0],[0,0,0,0],[9E+09,9E+09,9E+09,9E+09,9E+09,9E+09]];
  CONST robtarget Target_1850:=[[613.374984158,835.71563679,660.090342283],[0,0,1,0],[0,0,0,0],[9E+09,9E+09,9E+09,9E+09,9E+09,9E+09]];
  CONST robtarget Target_1860:=[[623.374984158,835.71563679,660.090342283],[0,0,1,0],[0,0,0,0],[9E+09,9E+09,9E+09,9E+09,9E+09,9E+09]];
  CONST robtarget Target_1870:=[[633.374984158,835.71563679,660.090342283],[0,0,1,0],[0,0,0,0],[9E+09,9E+09,9E+09,9E+09,9E+09,9E+09]];
  CONST robtarget Target_1880:=[[643.374984158,835.71563679,660.090342283],[0,0,1,0],[0,0,0,0],[9E+09,9E+09,9E+09,9E+09,9E+09,9E+09]];
  CONST robtarget Target_1890:=[[653.374984158,835.71563679,660.090342283],[0,0,1,0],[0,0,0,0],[9E+09,9E+09,9E+09,9E+09,9E+09,9E+09]];
  CONST robtarget Target_1900:=[[663.374984158,835.71563679,660.090342283],[0,0,1,0],[0,0,0,0],[9E+09,9E+09,9E+09,9E+09,9E+09,9E+09]];
  CONST robtarget Target_1910:=[[673.374984158,835.71563679,660.090342283],[0,0,1,0],[0,0,0,0],[9E+09,9E+09,9E+09,9E+09,9E+09,9E+09]];
  CONST robtarget Target_1920:=[[683.374984158,835.71563679,660.090342283],[0,0,1,0],[0,0,0,0],[9E+09,9E+09,9E+09,9E+09,9E+09,9E+09]];
  CONST robtarget Target_1930:=[[693.374984158,835.71563679,660.090342283],[0,0,1,0],[0,0,0,0],[9E+09,9E+09,9E+09,9E+09,9E+09,9E+09]];
  CONST robtarget Target_1940:=[[703.374984158,835.71563679,660.090342283],[0,0,1,0],[0,0,0,0],[9E+09,9E+09,9E+09,9E+09,9E+09,9E+09]];
  CONST robtarget Target_1950:=[[713.374984158,835.71563679,660.090342283],[0,0,1,0],[0,0,0,0],[9E+09,9E+09,9E+09,9E+09,9E+09,9E+09]];
  CONST robtarget Target_1960:=[[723.374984158,835.71563679,660.090342283],[0,0,1,0],[0,0,0,0],[9E+09,9E+09,9E+09,9E+09,9E+09,9E+09]];
  CONST robtarget Target_1970:=[[733.374984158,835.71563679,660.090342283],[0,0,1,0],[0,0,0,0],[9E+09,9E+09,9E+09,9E+09,9E+09,9E+09]];
  CONST robtarget Target_1980:=[[743.374984158,835.71563679,660.090342283],[0,0,1,0],[0,0,0,0],[9E+09,9E+09,9E+09,9E+09,9E+09,9E+09]];
  CONST robtarget Target_1990:=[[753.374984158,835.71563679,660.090342283],[0,0,1,0],[0,0,0,0],[9E+09,9E+09,9E+09,9E+09,9E+09,9E+09]];
  CONST robtarget Target_2000:=[[763.374984158,835.71563679,660.090342283],[0,0,1,0],[0,0,0,0],[9E+09,9E+09,9E+09,9E+09,9E+09,9E+09]];
  CONST robtarget Target_2010:=[[773.374984158,835.71563679,660.090342283],[0,0,1,0],[0,0,0,0],[9E+09,9E+09,9E+09,9E+09,9E+09,9E+09]];
  CONST robtarget Target_2020:=[[783.374984158,835.71563679,660.090342283],[0,0,1,0],[0,0,0,0],[9E+09,9E+09,9E+09,9E+09,9E+09,9E+09]];
  CONST robtarget Target_2030:=[[793.374984158,835.71563679,660.090342283],[0,0,1,0],[0,0,0,0],[9E+09,9E+09,9E+09,9E+09,9E+09,9E+09]];
  CONST robtarget Target_2040:=[[803.374984158,835.71563679,660.090342283],[0,0,1,0],[0,0,0,0],[9E+09,9E+09,9E+09,9E+09,9E+09,9E+09]];
  CONST robtarget Target_2050:=[[813.374984158,835.71563679,660.090342283],[0,0,1,0],[0,0,0,0],[9E+09,9E+09,9E+09,9E+09,9E+09,9E+09]];
  CONST robtarget Target_2060:=[[823.374984158,835.71563679,660.090342283],[0,0,1,0],[0,0,0,0],[9E+09,9E+09,9E+09,9E+09,9E+09,9E+09]];
  CONST robtarget Target_2070:=[[833.374984158,835.71563679,660.090342283],[0,0,1,0],[0,0,0,0],[9E+09,9E+09,9E+09,9E+09,9E+09,9E+09]];
  CONST robtarget Target_2080:=[[843.374984158,835.71563679,660.090342283],[0,0,1,0],[0,0,0,0],[9E+09,9E+09,9E+09,9E+09,9E+09,9E+09]];
  CONST robtarget Target_2090:=[[853.374984158,835.71563679,660.090342283],[0,0,1,0],[0,0,0,0],[9E+09,9E+09,9E+09,9E+09,9E+09,9E+09]];
  CONST robtarget Target_2100:=[[863.374984158,835.71563679,660.090342283],[0,0,1,0],[0,0,0,0],[9E+09,9E+09,9E+09,9E+09,9E+09,9E+09]];
  CONST robtarget Target_2110:=[[873.374984158,835.71563679,660.090342283],[0,0,1,0],[0,0,0,0],[9E+09,9E+09,9E+09,9E+09,9E+09,9E+09]];
  CONST robtarget Target_2120:=[[883.374984158,835.71563679,660.090342283],[0,0,1,0],[0,0,0,0],[9E+09,9E+09,9E+09,9E+09,9E+09,9E+09]];
  CONST robtarget Target_2130:=[[891.374984158,-133.68436321,660.090342283],[0,0,1,0],[0,0,0,0],[9E+09,9E+09,9E+09,9E+09,9E+09,9E+09]];
  CONST robtarget Target_2140:=[[891.374984158,-143.68436321,660.090342283],[0,0,1,0],[0,0,0,0],[9E+09,9E+09,9E+09,9E+09,9E+09,9E+09]];
  CONST robtarget Target_2150:=[[891.374984158,-153.68436321,660.090342283],[0,0,1,0],[0,0,0,0],[9E+09,9E+09,9E+09,9E+09,9E+09,9E+09]];
  CONST robtarget Target_2160:=[[891.374984158,-163.68436321,660.090342283],[0,0,1,0],[0,0,0,0],[9E+09,9E+09,9E+09,9E+09,9E+09,9E+09]];
  CONST robtarget Target_2170:=[[891.374984158,-173.68436321,660.090342283],[0,0,1,0],[0,0,0,0],[9E+09,9E+09,9E+09,9E+09,9E+09,9E+09]];
  CONST robtarget Target_2180:=[[891.374984158,-183.68436321,660.090342283],[0,0,1,0],[0,0,0,0],[9E+09,9E+09,9E+09,9E+09,9E+09,9E+09]];
  CONST robtarget Target_2190:=[[891.374984158,-193.68436321,660.090342283],[0,0,1,0],[0,0,0,0],[9E+09,9E+09,9E+09,9E+09,9E+09,9E+09]];
  CONST robtarget Target_2200:=[[891.374984158,-203.68436321,660.090342283],[0,0,1,0],[0,0,0,0],[9E+09,9E+09,9E+09,9E+09,9E+09,9E+09]];
  CONST robtarget Target_2210:=[[891.374984158,-213.68436321,660.090342283],[0,0,1,0],[0,0,0,0],[9E+09,9E+09,9E+09,9E+09,9E+09,9E+09]];
  CONST robtarget Target_2220:=[[891.374984158,-223.68436321,660.090342283],[0,0,1,0],[0,0,0,0],[9E+09,9E+09,9E+09,9E+09,9E+09,9E+09]];
  CONST robtarget Target_2230:=[[891.374984158,-233.68436321,660.090342283],[0,0,1,0],[0,0,0,0],[9E+09,9E+09,9E+09,9E+09,9E+09,9E+09]];
  CONST robtarget Target_2240:=[[891.374984158,-243.68436321,660.090342283],[0,0,1,0],[0,0,0,0],[9E+09,9E+09,9E+09,9E+09,9E+09,9E+09]];
  CONST robtarget Target_2250:=[[891.374984158,-253.68436321,660.090342283],[0,0,1,0],[0,0,0,0],[9E+09,9E+09,9E+09,9E+09,9E+09,9E+09]];
  CONST robtarget Target_2260:=[[891.374984158,-263.68436321,660.090342283],[0,0,1,0],[0,0,0,0],[9E+09,9E+09,9E+09,9E+09,9E+09,9E+09]];
  CONST robtarget Target_2270:=[[891.374984158,-273.68436321,660.090342283],[0,0,1,0],[0,0,0,0],[9E+09,9E+09,9E+09,9E+09,9E+09,9E+09]];
  CONST robtarget Target_2280:=[[891.374984158,-283.68436321,660.090342283],[0,0,1,0],[0,0,0,0],[9E+09,9E+09,9E+09,9E+09,9E+09,9E+09]];
  CONST robtarget Target_2290:=[[891.374984158,-293.68436321,660.090342283],[0,0,1,0],[0,0,0,0],[9E+09,9E+09,9E+09,9E+09,9E+09,9E+09]];
  CONST robtarget Target_2300:=[[891.374984158,-303.68436321,660.090342283],[0,0,1,0],[0,0,0,0],[9E+09,9E+09,9E+09,9E+09,9E+09,9E+09]];
  CONST robtarget Target_2310:=[[891.374984158,-313.68436321,660.090342283],[0,0,1,0],[0,0,0,0],[9E+09,9E+09,9E+09,9E+09,9E+09,9E+09]];
  CONST robtarget Target_2320:=[[891.374984158,-323.68436321,660.090342283],[0,0,1,0],[0,0,0,0],[9E+09,9E+09,9E+09,9E+09,9E+09,9E+09]];
  CONST robtarget Target_2330:=[[891.374984158,-333.68436321,660.090342283],[0,0,1,0],[0,0,0,0],[9E+09,9E+09,9E+09,9E+09,9E+09,9E+09]];
  CONST robtarget Target_2340:=[[891.374984158,-343.68436321,660.090342283],[0,0,1,0],[0,0,0,0],[9E+09,9E+09,9E+09,9E+09,9E+09,9E+09]];
  CONST robtarget Target_2350:=[[891.374984158,-353.68436321,660.090342283],[0,0,1,0],[0,0,0,0],[9E+09,9E+09,9E+09,9E+09,9E+09,9E+09]];
  CONST robtarget Target_2360:=[[891.374984158,-363.68436321,660.090342283],[0,0,1,0],[0,0,0,0],[9E+09,9E+09,9E+09,9E+09,9E+09,9E+09]];
  CONST robtarget Target_2370:=[[891.374984158,-373.68436321,660.090342283],[0,0,1,0],[0,0,0,0],[9E+09,9E+09,9E+09,9E+09,9E+09,9E+09]];
  CONST robtarget Target_2380:=[[891.374984158,-383.68436321,660.090342283],[0,0,1,0],[0,0,0,0],[9E+09,9E+09,9E+09,9E+09,9E+09,9E+09]];
  CONST robtarget Target_2390:=[[891.374984158,-393.68436321,660.090342283],[0,0,1,0],[0,0,0,0],[9E+09,9E+09,9E+09,9E+09,9E+09,9E+09]];
  CONST robtarget Target_2400:=[[891.374984158,-403.68436321,660.090342283],[0,0,1,0],[0,0,0,0],[9E+09,9E+09,9E+09,9E+09,9E+09,9E+09]];
  CONST robtarget Target_2410:=[[891.374984158,-413.68436321,660.090342283],[0,0,1,0],[0,0,0,0],[9E+09,9E+09,9E+09,9E+09,9E+09,9E+09]];
  CONST robtarget Target_2420:=[[891.374984158,-423.68436321,660.090342283],[0,0,1,0],[0,0,0,0],[9E+09,9E+09,9E+09,9E+09,9E+09,9E+09]];
  CONST robtarget Target_2430:=[[891.374984158,-433.68436321,660.090342283],[0,0,1,0],[0,0,0,0],[9E+09,9E+09,9E+09,9E+09,9E+09,9E+09]];
  CONST robtarget Target_2440:=[[891.374984158,-443.68436321,660.090342283],[0,0,1,0],[0,0,0,0],[9E+09,9E+09,9E+09,9E+09,9E+09,9E+09]];
  CONST robtarget Target_2450:=[[891.374984158,-453.68436321,660.090342283],[0,0,1,0],[0,0,0,0],[9E+09,9E+09,9E+09,9E+09,9E+09,9E+09]];
  CONST robtarget Target_2460:=[[891.374984158,-463.68436321,660.090342283],[0,0,1,0],[0,0,0,0],[9E+09,9E+09,9E+09,9E+09,9E+09,9E+09]];
  CONST robtarget Target_2470:=[[891.374984158,-473.68436321,660.090342283],[0,0,1,0],[0,0,0,0],[9E+09,9E+09,9E+09,9E+09,9E+09,9E+09]];
  CONST robtarget Target_2480:=[[891.374984158,-483.68436321,660.090342283],[0,0,1,0],[0,0,0,0],[9E+09,9E+09,9E+09,9E+09,9E+09,9E+09]];
  CONST robtarget Target_2490:=[[891.374984158,-493.68436321,660.090342283],[0,0,1,0],[0,0,0,0],[9E+09,9E+09,9E+09,9E+09,9E+09,9E+09]];
  CONST robtarget Target_2500:=[[891.374984158,-503.68436321,660.090342283],[0,0,1,0],[0,0,0,0],[9E+09,9E+09,9E+09,9E+09,9E+09,9E+09]];
  CONST robtarget Target_2510:=[[891.374984158,-513.68436321,660.090342283],[0,0,1,0],[0,0,0,0],[9E+09,9E+09,9E+09,9E+09,9E+09,9E+09]];
  CONST robtarget Target_2520:=[[891.374984158,-523.68436321,660.090342283],[0,0,1,0],[0,0,0,0],[9E+09,9E+09,9E+09,9E+09,9E+09,9E+09]];
  CONST robtarget Target_2530:=[[891.374984158,-533.68436321,660.090342283],[0,0,1,0],[0,0,0,0],[9E+09,9E+09,9E+09,9E+09,9E+09,9E+09]];
  CONST robtarget Target_2540:=[[891.374984158,-543.68436321,660.090342283],[0,0,1,0],[0,0,0,0],[9E+09,9E+09,9E+09,9E+09,9E+09,9E+09]];
  CONST robtarget Target_2550:=[[891.374984158,-553.68436321,660.090342283],[0,0,1,0],[0,0,0,0],[9E+09,9E+09,9E+09,9E+09,9E+09,9E+09]];
  CONST robtarget Target_2560:=[[891.374984158,-563.68436321,660.090342283],[0,0,1,0],[0,0,0,0],[9E+09,9E+09,9E+09,9E+09,9E+09,9E+09]];
  CONST robtarget Target_2570:=[[891.374984158,-573.68436321,660.090342283],[0,0,1,0],[0,0,0,0],[9E+09,9E+09,9E+09,9E+09,9E+09,9E+09]];
  CONST robtarget Target_2580:=[[373.374984158,352.91563679,660.090342283],[0,0,1,0],[0,0,0,0],[9E+09,9E+09,9E+09,9E+09,9E+09,9E+09]];
  CONST robtarget Target_2590:=[[373.374984158,342.91563679,660.090342283],[0,0,1,0],[0,0,0,0],[9E+09,9E+09,9E+09,9E+09,9E+09,9E+09]];
  CONST robtarget Target_2600:=[[373.374984158,332.91563679,660.090342283],[0,0,1,0],[0,0,0,0],[9E+09,9E+09,9E+09,9E+09,9E+09,9E+09]];
  CONST robtarget Target_2610:=[[373.374984158,322.91563679,660.090342283],[0,0,1,0],[0,0,0,0],[9E+09,9E+09,9E+09,9E+09,9E+09,9E+09]];
  CONST robtarget Target_2620:=[[373.374984158,312.91563679,660.090342283],[0,0,1,0],[0,0,0,0],[9E+09,9E+09,9E+09,9E+09,9E+09,9E+09]];
  CONST robtarget Target_2630:=[[373.374984158,302.91563679,660.090342283],[0,0,1,0],[0,0,0,0],[9E+09,9E+09,9E+09,9E+09,9E+09,9E+09]];
  CONST robtarget Target_2640:=[[373.374984158,292.91563679,660.090342283],[0,0,1,0],[0,0,0,0],[9E+09,9E+09,9E+09,9E+09,9E+09,9E+09]];
  CONST robtarget Target_2650:=[[373.374984158,282.91563679,660.090342283],[0,0,1,0],[0,0,0,0],[9E+09,9E+09,9E+09,9E+09,9E+09,9E+09]];
  CONST robtarget Target_2660:=[[373.374984158,272.91563679,660.090342283],[0,0,1,0],[0,0,0,0],[9E+09,9E+09,9E+09,9E+09,9E+09,9E+09]];
  CONST robtarget Target_2670:=[[373.374984158,262.91563679,660.090342283],[0,0,1,0],[0,0,0,0],[9E+09,9E+09,9E+09,9E+09,9E+09,9E+09]];
  CONST robtarget Target_2680:=[[373.374984158,252.91563679,660.090342283],[0,0,1,0],[0,0,0,0],[9E+09,9E+09,9E+09,9E+09,9E+09,9E+09]];
  CONST robtarget Target_2690:=[[373.374984158,242.91563679,660.090342283],[0,0,1,0],[0,0,0,0],[9E+09,9E+09,9E+09,9E+09,9E+09,9E+09]];
  CONST robtarget Target_2700:=[[373.374984158,232.91563679,660.090342283],[0,0,1,0],[0,0,0,0],[9E+09,9E+09,9E+09,9E+09,9E+09,9E+09]];
  CONST robtarget Target_2710:=[[373.374984158,222.91563679,660.090342283],[0,0,1,0],[0,0,0,0],[9E+09,9E+09,9E+09,9E+09,9E+09,9E+09]];
  CONST robtarget Target_2720:=[[373.374984158,212.91563679,660.090342283],[0,0,1,0],[0,0,0,0],[9E+09,9E+09,9E+09,9E+09,9E+09,9E+09]];
  CONST robtarget Target_2730:=[[373.374984158,202.91563679,660.090342283],[0,0,1,0],[0,0,0,0],[9E+09,9E+09,9E+09,9E+09,9E+09,9E+09]];
  CONST robtarget Target_2740:=[[373.374984158,192.91563679,660.090342283],[0,0,1,0],[0,0,0,0],[9E+09,9E+09,9E+09,9E+09,9E+09,9E+09]];
  CONST robtarget Target_2750:=[[373.374984158,182.91563679,660.090342283],[0,0,1,0],[0,0,0,0],[9E+09,9E+09,9E+09,9E+09,9E+09,9E+09]];
  CONST robtarget Target_2760:=[[373.374984158,172.91563679,660.090342283],[0,0,1,0],[0,0,0,0],[9E+09,9E+09,9E+09,9E+09,9E+09,9E+09]];
  CONST robtarget Target_2770:=[[373.374984158,162.91563679,660.090342283],[0,0,1,0],[0,0,0,0],[9E+09,9E+09,9E+09,9E+09,9E+09,9E+09]];
  CONST robtarget Target_2780:=[[373.374984158,152.91563679,660.090342283],[0,0,1,0],[0,0,0,0],[9E+09,9E+09,9E+09,9E+09,9E+09,9E+09]];
  CONST robtarget Target_2790:=[[373.374984158,142.91563679,660.090342283],[0,0,1,0],[0,0,0,0],[9E+09,9E+09,9E+09,9E+09,9E+09,9E+09]];
  CONST robtarget Target_2800:=[[373.374984158,132.91563679,660.090342283],[0,0,1,0],[0,0,0,0],[9E+09,9E+09,9E+09,9E+09,9E+09,9E+09]];
  CONST robtarget Target_2810:=[[373.374984158,122.91563679,660.090342283],[0,0,1,0],[0,0,0,0],[9E+09,9E+09,9E+09,9E+09,9E+09,9E+09]];
  CONST robtarget Target_2820:=[[373.374984158,112.91563679,660.090342283],[0,0,1,0],[0,0,0,0],[9E+09,9E+09,9E+09,9E+09,9E+09,9E+09]];
  CONST robtarget Target_2830:=[[373.374984158,102.91563679,660.090342283],[0,0,1,0],[0,0,0,0],[9E+09,9E+09,9E+09,9E+09,9E+09,9E+09]];
  CONST robtarget Target_2840:=[[373.374984158,92.91563679,660.090342283],[0,0,1,0],[0,0,0,0],[9E+09,9E+09,9E+09,9E+09,9E+09,9E+09]];
  CONST robtarget Target_2850:=[[373.374984158,82.91563679,660.090342283],[0,0,1,0],[0,0,0,0],[9E+09,9E+09,9E+09,9E+09,9E+09,9E+09]];
  CONST robtarget Target_2860:=[[373.374984158,72.91563679,660.090342283],[0,0,1,0],[0,0,0,0],[9E+09,9E+09,9E+09,9E+09,9E+09,9E+09]];
  CONST robtarget Target_2870:=[[373.374984158,62.91563679,660.090342283],[0,0,1,0],[0,0,0,0],[9E+09,9E+09,9E+09,9E+09,9E+09,9E+09]];
  CONST robtarget Target_2880:=[[373.374984158,52.91563679,660.090342283],[0,0,1,0],[0,0,0,0],[9E+09,9E+09,9E+09,9E+09,9E+09,9E+09]];
  CONST robtarget Target_2890:=[[373.374984158,42.91563679,660.090342283],[0,0,1,0],[0,0,0,0],[9E+09,9E+09,9E+09,9E+09,9E+09,9E+09]];
  CONST robtarget Target_2900:=[[373.374984158,32.91563679,660.090342283],[0,0,1,0],[0,0,0,0],[9E+09,9E+09,9E+09,9E+09,9E+09,9E+09]];
  CONST robtarget Target_2910:=[[373.374984158,22.91563679,660.090342283],[0,0,1,0],[0,0,0,0],[9E+09,9E+09,9E+09,9E+09,9E+09,9E+09]];
  CONST robtarget Target_2920:=[[373.374984158,12.91563679,660.090342283],[0,0,1,0],[0,0,0,0],[9E+09,9E+09,9E+09,9E+09,9E+09,9E+09]];
  CONST robtarget Target_2930:=[[373.374984158,2.91563679,660.090342283],[0,0,1,0],[0,0,0,0],[9E+09,9E+09,9E+09,9E+09,9E+09,9E+09]];
  CONST robtarget Target_2940:=[[373.374984158,-7.08436321,660.090342283],[0,0,1,0],[0,0,0,0],[9E+09,9E+09,9E+09,9E+09,9E+09,9E+09]];
  CONST robtarget Target_2950:=[[373.374984158,-17.08436321,660.090342283],[0,0,1,0],[0,0,0,0],[9E+09,9E+09,9E+09,9E+09,9E+09,9E+09]];
  CONST robtarget Target_2960:=[[373.374984158,-27.08436321,660.090342283],[0,0,1,0],[0,0,0,0],[9E+09,9E+09,9E+09,9E+09,9E+09,9E+09]];
  CONST robtarget Target_2970:=[[373.374984158,-37.08436321,660.090342283],[0,0,1,0],[0,0,0,0],[9E+09,9E+09,9E+09,9E+09,9E+09,9E+09]];
  CONST robtarget Target_2980:=[[373.374984158,-47.08436321,660.090342283],[0,0,1,0],[0,0,0,0],[9E+09,9E+09,9E+09,9E+09,9E+09,9E+09]];
  CONST robtarget Target_2990:=[[373.374984158,-57.08436321,660.090342283],[0,0,1,0],[0,0,0,0],[9E+09,9E+09,9E+09,9E+09,9E+09,9E+09]];
  CONST robtarget Target_3000:=[[373.374984158,-67.08436321,660.090342283],[0,0,1,0],[0,0,0,0],[9E+09,9E+09,9E+09,9E+09,9E+09,9E+09]];
  CONST robtarget Target_3010:=[[373.374984158,-77.08436321,660.090342283],[0,0,1,0],[0,0,0,0],[9E+09,9E+09,9E+09,9E+09,9E+09,9E+09]];
  CONST robtarget Target_3020:=[[373.374984158,-87.08436321,660.090342283],[0,0,1,0],[0,0,0,0],[9E+09,9E+09,9E+09,9E+09,9E+09,9E+09]];
  CONST robtarget Target_3030:=[[891.374984158,837.71563679,660.090342283],[0,0,1,0],[0,0,0,0],[9E+09,9E+09,9E+09,9E+09,9E+09,9E+09]];
  CONST robtarget Target_3040:=[[891.374984158,827.71563679,660.090342283],[0,0,1,0],[0,0,0,0],[9E+09,9E+09,9E+09,9E+09,9E+09,9E+09]];
  CONST robtarget Target_3050:=[[891.374984158,817.71563679,660.090342283],[0,0,1,0],[0,0,0,0],[9E+09,9E+09,9E+09,9E+09,9E+09,9E+09]];
  CONST robtarget Target_3060:=[[891.374984158,807.71563679,660.090342283],[0,0,1,0],[0,0,0,0],[9E+09,9E+09,9E+09,9E+09,9E+09,9E+09]];
  CONST robtarget Target_3070:=[[891.374984158,797.71563679,660.090342283],[0,0,1,0],[0,0,0,0],[9E+09,9E+09,9E+09,9E+09,9E+09,9E+09]];
  CONST robtarget Target_3080:=[[891.374984158,787.71563679,660.090342283],[0,0,1,0],[0,0,0,0],[9E+09,9E+09,9E+09,9E+09,9E+09,9E+09]];
  CONST robtarget Target_3090:=[[891.374984158,777.71563679,660.090342283],[0,0,1,0],[0,0,0,0],[9E+09,9E+09,9E+09,9E+09,9E+09,9E+09]];
  CONST robtarget Target_3100:=[[891.374984158,767.71563679,660.090342283],[0,0,1,0],[0,0,0,0],[9E+09,9E+09,9E+09,9E+09,9E+09,9E+09]];
  CONST robtarget Target_3110:=[[891.374984158,757.71563679,660.090342283],[0,0,1,0],[0,0,0,0],[9E+09,9E+09,9E+09,9E+09,9E+09,9E+09]];
  CONST robtarget Target_3120:=[[891.374984158,747.71563679,660.090342283],[0,0,1,0],[0,0,0,0],[9E+09,9E+09,9E+09,9E+09,9E+09,9E+09]];
  CONST robtarget Target_3130:=[[891.374984158,737.71563679,660.090342283],[0,0,1,0],[0,0,0,0],[9E+09,9E+09,9E+09,9E+09,9E+09,9E+09]];
  CONST robtarget Target_3140:=[[891.374984158,727.71563679,660.090342283],[0,0,1,0],[0,0,0,0],[9E+09,9E+09,9E+09,9E+09,9E+09,9E+09]];
  CONST robtarget Target_3150:=[[891.374984158,717.71563679,660.090342283],[0,0,1,0],[0,0,0,0],[9E+09,9E+09,9E+09,9E+09,9E+09,9E+09]];
  CONST robtarget Target_3160:=[[891.374984158,707.71563679,660.090342283],[0,0,1,0],[0,0,0,0],[9E+09,9E+09,9E+09,9E+09,9E+09,9E+09]];
  CONST robtarget Target_3170:=[[891.374984158,697.71563679,660.090342283],[0,0,1,0],[0,0,0,0],[9E+09,9E+09,9E+09,9E+09,9E+09,9E+09]];
  CONST robtarget Target_3180:=[[891.374984158,687.71563679,660.090342283],[0,0,1,0],[0,0,0,0],[9E+09,9E+09,9E+09,9E+09,9E+09,9E+09]];
  CONST robtarget Target_3190:=[[891.374984158,677.71563679,660.090342283],[0,0,1,0],[0,0,0,0],[9E+09,9E+09,9E+09,9E+09,9E+09,9E+09]];
  CONST robtarget Target_3200:=[[891.374984158,667.71563679,660.090342283],[0,0,1,0],[0,0,0,0],[9E+09,9E+09,9E+09,9E+09,9E+09,9E+09]];
  CONST robtarget Target_3210:=[[891.374984158,657.71563679,660.090342283],[0,0,1,0],[0,0,0,0],[9E+09,9E+09,9E+09,9E+09,9E+09,9E+09]];
  CONST robtarget Target_3220:=[[891.374984158,647.71563679,660.090342283],[0,0,1,0],[0,0,0,0],[9E+09,9E+09,9E+09,9E+09,9E+09,9E+09]];
  CONST robtarget Target_3230:=[[891.374984158,637.71563679,660.090342283],[0,0,1,0],[0,0,0,0],[9E+09,9E+09,9E+09,9E+09,9E+09,9E+09]];
  CONST robtarget Target_3240:=[[891.374984158,627.71563679,660.090342283],[0,0,1,0],[0,0,0,0],[9E+09,9E+09,9E+09,9E+09,9E+09,9E+09]];
  CONST robtarget Target_3250:=[[891.374984158,617.71563679,660.090342283],[0,0,1,0],[0,0,0,0],[9E+09,9E+09,9E+09,9E+09,9E+09,9E+09]];
  CONST robtarget Target_3260:=[[891.374984158,607.71563679,660.090342283],[0,0,1,0],[0,0,0,0],[9E+09,9E+09,9E+09,9E+09,9E+09,9E+09]];
  CONST robtarget Target_3270:=[[891.374984158,597.71563679,660.090342283],[0,0,1,0],[0,0,0,0],[9E+09,9E+09,9E+09,9E+09,9E+09,9E+09]];
  CONST robtarget Target_3280:=[[891.374984158,587.71563679,660.090342283],[0,0,1,0],[0,0,0,0],[9E+09,9E+09,9E+09,9E+09,9E+09,9E+09]];
  CONST robtarget Target_3290:=[[891.374984158,577.71563679,660.090342283],[0,0,1,0],[0,0,0,0],[9E+09,9E+09,9E+09,9E+09,9E+09,9E+09]];
  CONST robtarget Target_3300:=[[891.374984158,567.71563679,660.090342283],[0,0,1,0],[0,0,0,0],[9E+09,9E+09,9E+09,9E+09,9E+09,9E+09]];
  CONST robtarget Target_3310:=[[891.374984158,557.71563679,660.090342283],[0,0,1,0],[0,0,0,0],[9E+09,9E+09,9E+09,9E+09,9E+09,9E+09]];
  CONST robtarget Target_3320:=[[891.374984158,547.71563679,660.090342283],[0,0,1,0],[0,0,0,0],[9E+09,9E+09,9E+09,9E+09,9E+09,9E+09]];
  CONST robtarget Target_3330:=[[891.374984158,537.71563679,660.090342283],[0,0,1,0],[0,0,0,0],[9E+09,9E+09,9E+09,9E+09,9E+09,9E+09]];
  CONST robtarget Target_3340:=[[891.374984158,527.71563679,660.090342283],[0,0,1,0],[0,0,0,0],[9E+09,9E+09,9E+09,9E+09,9E+09,9E+09]];
  CONST robtarget Target_3350:=[[891.374984158,517.71563679,660.090342283],[0,0,1,0],[0,0,0,0],[9E+09,9E+09,9E+09,9E+09,9E+09,9E+09]];
  CONST robtarget Target_3360:=[[891.374984158,507.71563679,660.090342283],[0,0,1,0],[0,0,0,0],[9E+09,9E+09,9E+09,9E+09,9E+09,9E+09]];
  CONST robtarget Target_3370:=[[891.374984158,497.71563679,660.090342283],[0,0,1,0],[0,0,0,0],[9E+09,9E+09,9E+09,9E+09,9E+09,9E+09]];
  CONST robtarget Target_3380:=[[891.374984158,487.71563679,660.090342283],[0,0,1,0],[0,0,0,0],[9E+09,9E+09,9E+09,9E+09,9E+09,9E+09]];
  CONST robtarget Target_3390:=[[891.374984158,477.71563679,660.090342283],[0,0,1,0],[0,0,0,0],[9E+09,9E+09,9E+09,9E+09,9E+09,9E+09]];
  CONST robtarget Target_3400:=[[891.374984158,467.71563679,660.090342283],[0,0,1,0],[0,0,0,0],[9E+09,9E+09,9E+09,9E+09,9E+09,9E+09]];
  CONST robtarget Target_3410:=[[891.374984158,457.71563679,660.090342283],[0,0,1,0],[0,0,0,0],[9E+09,9E+09,9E+09,9E+09,9E+09,9E+09]];
  CONST robtarget Target_3420:=[[891.374984158,447.71563679,660.090342283],[0,0,1,0],[0,0,0,0],[9E+09,9E+09,9E+09,9E+09,9E+09,9E+09]];
  CONST robtarget Target_3430:=[[891.374984158,437.71563679,660.090342283],[0,0,1,0],[0,0,0,0],[9E+09,9E+09,9E+09,9E+09,9E+09,9E+09]];
  CONST robtarget Target_3440:=[[891.374984158,427.71563679,660.090342283],[0,0,1,0],[0,0,0,0],[9E+09,9E+09,9E+09,9E+09,9E+09,9E+09]];
  CONST robtarget Target_3450:=[[891.374984158,417.71563679,660.090342283],[0,0,1,0],[0,0,0,0],[9E+09,9E+09,9E+09,9E+09,9E+09,9E+09]];
  CONST robtarget Target_3460:=[[891.374984158,407.71563679,660.090342283],[0,0,1,0],[0,0,0,0],[9E+09,9E+09,9E+09,9E+09,9E+09,9E+09]];
  CONST robtarget Target_3470:=[[891.374984158,397.71563679,660.090342283],[0,0,1,0],[0,0,0,0],[9E+09,9E+09,9E+09,9E+09,9E+09,9E+09]];
  CONST robtarget Target_3480:=[[373.374984158,837.71563679,660.090342283],[0,0,1,0],[0,0,0,0],[9E+09,9E+09,9E+09,9E+09,9E+09,9E+09]];
  CONST robtarget Target_3490:=[[373.374984158,827.71563679,660.090342283],[0,0,1,0],[0,0,0,0],[9E+09,9E+09,9E+09,9E+09,9E+09,9E+09]];
  CONST robtarget Target_3500:=[[373.374984158,817.71563679,660.090342283],[0,0,1,0],[0,0,0,0],[9E+09,9E+09,9E+09,9E+09,9E+09,9E+09]];
  CONST robtarget Target_3510:=[[373.374984158,807.71563679,660.090342283],[0,0,1,0],[0,0,0,0],[9E+09,9E+09,9E+09,9E+09,9E+09,9E+09]];
  CONST robtarget Target_3520:=[[373.374984158,797.71563679,660.090342283],[0,0,1,0],[0,0,0,0],[9E+09,9E+09,9E+09,9E+09,9E+09,9E+09]];
  CONST robtarget Target_3530:=[[373.374984158,787.71563679,660.090342283],[0,0,1,0],[0,0,0,0],[9E+09,9E+09,9E+09,9E+09,9E+09,9E+09]];
  CONST robtarget Target_3540:=[[373.374984158,777.71563679,660.090342283],[0,0,1,0],[0,0,0,0],[9E+09,9E+09,9E+09,9E+09,9E+09,9E+09]];
  CONST robtarget Target_3550:=[[373.374984158,767.71563679,660.090342283],[0,0,1,0],[0,0,0,0],[9E+09,9E+09,9E+09,9E+09,9E+09,9E+09]];
  CONST robtarget Target_3560:=[[373.374984158,757.71563679,660.090342283],[0,0,1,0],[0,0,0,0],[9E+09,9E+09,9E+09,9E+09,9E+09,9E+09]];
  CONST robtarget Target_3570:=[[373.374984158,747.71563679,660.090342283],[0,0,1,0],[0,0,0,0],[9E+09,9E+09,9E+09,9E+09,9E+09,9E+09]];
  CONST robtarget Target_3580:=[[373.374984158,737.71563679,660.090342283],[0,0,1,0],[0,0,0,0],[9E+09,9E+09,9E+09,9E+09,9E+09,9E+09]];
  CONST robtarget Target_3590:=[[373.374984158,727.71563679,660.090342283],[0,0,1,0],[0,0,0,0],[9E+09,9E+09,9E+09,9E+09,9E+09,9E+09]];
  CONST robtarget Target_3600:=[[373.374984158,717.71563679,660.090342283],[0,0,1,0],[0,0,0,0],[9E+09,9E+09,9E+09,9E+09,9E+09,9E+09]];
  CONST robtarget Target_3610:=[[373.374984158,707.71563679,660.090342283],[0,0,1,0],[0,0,0,0],[9E+09,9E+09,9E+09,9E+09,9E+09,9E+09]];
  CONST robtarget Target_3620:=[[373.374984158,697.71563679,660.090342283],[0,0,1,0],[0,0,0,0],[9E+09,9E+09,9E+09,9E+09,9E+09,9E+09]];
  CONST robtarget Target_3630:=[[373.374984158,687.71563679,660.090342283],[0,0,1,0],[0,0,0,0],[9E+09,9E+09,9E+09,9E+09,9E+09,9E+09]];
  CONST robtarget Target_3640:=[[373.374984158,677.71563679,660.090342283],[0,0,1,0],[0,0,0,0],[9E+09,9E+09,9E+09,9E+09,9E+09,9E+09]];
  CONST robtarget Target_3650:=[[373.374984158,667.71563679,660.090342283],[0,0,1,0],[0,0,0,0],[9E+09,9E+09,9E+09,9E+09,9E+09,9E+09]];
  CONST robtarget Target_3660:=[[373.374984158,657.71563679,660.090342283],[0,0,1,0],[0,0,0,0],[9E+09,9E+09,9E+09,9E+09,9E+09,9E+09]];
  CONST robtarget Target_3670:=[[373.374984158,647.71563679,660.090342283],[0,0,1,0],[0,0,0,0],[9E+09,9E+09,9E+09,9E+09,9E+09,9E+09]];
  CONST robtarget Target_3680:=[[373.374984158,637.71563679,660.090342283],[0,0,1,0],[0,0,0,0],[9E+09,9E+09,9E+09,9E+09,9E+09,9E+09]];
  CONST robtarget Target_3690:=[[373.374984158,627.71563679,660.090342283],[0,0,1,0],[0,0,0,0],[9E+09,9E+09,9E+09,9E+09,9E+09,9E+09]];
  CONST robtarget Target_3700:=[[373.374984158,617.71563679,660.090342283],[0,0,1,0],[0,0,0,0],[9E+09,9E+09,9E+09,9E+09,9E+09,9E+09]];
  CONST robtarget Target_3710:=[[373.374984158,607.71563679,660.090342283],[0,0,1,0],[0,0,0,0],[9E+09,9E+09,9E+09,9E+09,9E+09,9E+09]];
  CONST robtarget Target_3720:=[[373.374984158,597.71563679,660.090342283],[0,0,1,0],[0,0,0,0],[9E+09,9E+09,9E+09,9E+09,9E+09,9E+09]];
  CONST robtarget Target_3730:=[[373.374984158,587.71563679,660.090342283],[0,0,1,0],[0,0,0,0],[9E+09,9E+09,9E+09,9E+09,9E+09,9E+09]];
  CONST robtarget Target_3740:=[[373.374984158,577.71563679,660.090342283],[0,0,1,0],[0,0,0,0],[9E+09,9E+09,9E+09,9E+09,9E+09,9E+09]];
  CONST robtarget Target_3750:=[[373.374984158,567.71563679,660.090342283],[0,0,1,0],[0,0,0,0],[9E+09,9E+09,9E+09,9E+09,9E+09,9E+09]];
  CONST robtarget Target_3760:=[[373.374984158,557.71563679,660.090342283],[0,0,1,0],[0,0,0,0],[9E+09,9E+09,9E+09,9E+09,9E+09,9E+09]];
  CONST robtarget Target_3770:=[[373.374984158,547.71563679,660.090342283],[0,0,1,0],[0,0,0,0],[9E+09,9E+09,9E+09,9E+09,9E+09,9E+09]];
  CONST robtarget Target_3780:=[[373.374984158,537.71563679,660.090342283],[0,0,1,0],[0,0,0,0],[9E+09,9E+09,9E+09,9E+09,9E+09,9E+09]];
  CONST robtarget Target_3790:=[[373.374984158,527.71563679,660.090342283],[0,0,1,0],[0,0,0,0],[9E+09,9E+09,9E+09,9E+09,9E+09,9E+09]];
  CONST robtarget Target_3800:=[[373.374984158,517.71563679,660.090342283],[0,0,1,0],[0,0,0,0],[9E+09,9E+09,9E+09,9E+09,9E+09,9E+09]];
  CONST robtarget Target_3810:=[[373.374984158,507.71563679,660.090342283],[0,0,1,0],[0,0,0,0],[9E+09,9E+09,9E+09,9E+09,9E+09,9E+09]];
  CONST robtarget Target_3820:=[[373.374984158,497.71563679,660.090342283],[0,0,1,0],[0,0,0,0],[9E+09,9E+09,9E+09,9E+09,9E+09,9E+09]];
  CONST robtarget Target_3830:=[[373.374984158,487.71563679,660.090342283],[0,0,1,0],[0,0,0,0],[9E+09,9E+09,9E+09,9E+09,9E+09,9E+09]];
  CONST robtarget Target_3840:=[[373.374984158,477.71563679,660.090342283],[0,0,1,0],[0,0,0,0],[9E+09,9E+09,9E+09,9E+09,9E+09,9E+09]];
  CONST robtarget Target_3850:=[[373.374984158,467.71563679,660.090342283],[0,0,1,0],[0,0,0,0],[9E+09,9E+09,9E+09,9E+09,9E+09,9E+09]];
  CONST robtarget Target_3860:=[[373.374984158,457.71563679,660.090342283],[0,0,1,0],[0,0,0,0],[9E+09,9E+09,9E+09,9E+09,9E+09,9E+09]];
  CONST robtarget Target_3870:=[[373.374984158,447.71563679,660.090342283],[0,0,1,0],[0,0,0,0],[9E+09,9E+09,9E+09,9E+09,9E+09,9E+09]];
  CONST robtarget Target_3880:=[[373.374984158,437.71563679,660.090342283],[0,0,1,0],[0,0,0,0],[9E+09,9E+09,9E+09,9E+09,9E+09,9E+09]];
  CONST robtarget Target_3890:=[[373.374984158,427.71563679,660.090342283],[0,0,1,0],[0,0,0,0],[9E+09,9E+09,9E+09,9E+09,9E+09,9E+09]];
  CONST robtarget Target_3900:=[[373.374984158,417.71563679,660.090342283],[0,0,1,0],[0,0,0,0],[9E+09,9E+09,9E+09,9E+09,9E+09,9E+09]];
  CONST robtarget Target_3910:=[[373.374984158,407.71563679,660.090342283],[0,0,1,0],[0,0,0,0],[9E+09,9E+09,9E+09,9E+09,9E+09,9E+09]];
  CONST robtarget Target_3920:=[[373.374984158,397.71563679,660.090342283],[0,0,1,0],[0,0,0,0],[9E+09,9E+09,9E+09,9E+09,9E+09,9E+09]];
  CONST robtarget Target_3930:=[[373.374963375,397.715599785,811.779393568],[0.000000059,-0.00000001,1,-0.000000019],[0,-1,0,0],[9E+09,9E+09,9E+09,9E+09,9E+09,9E+09]];
  CONST robtarget Target_3940:=[[605.756953612,397.715613811,811.779394215],[0.00000009,-0.000000014,1,0.000000006],[0,-1,0,0],[9E+09,9E+09,9E+09,9E+09,9E+09,9E+09]];
  CONST robtarget Target_3950:=[[885.457956562,397.715597071,811.779409936],[0.000000132,-0.000000025,1,-0.000000004],[0,-1,0,0],[9E+09,9E+09,9E+09,9E+09,9E+09,9E+09]];
  CONST robtarget Target_3960:=[[885.457954174,345.735297458,693.687988495],[0,0,1,0],[0,-1,0,0],[9E+09,9E+09,9E+09,9E+09,9E+09,9E+09]];
  CONST robtarget Target_3970:=[[891.374984158,352.91563679,660.090342283],[0,0,1,0],[0,0,0,0],[9E+09,9E+09,9E+09,9E+09,9E+09,9E+09]];
  CONST robtarget Target_3980:=[[891.374984158,342.91563679,660.090342283],[0,0,1,0],[0,0,0,0],[9E+09,9E+09,9E+09,9E+09,9E+09,9E+09]];
  CONST robtarget Target_3990:=[[891.374984158,332.91563679,660.090342283],[0,0,1,0],[0,0,0,0],[9E+09,9E+09,9E+09,9E+09,9E+09,9E+09]];
  CONST robtarget Target_4000:=[[891.374984158,322.91563679,660.090342283],[0,0,1,0],[0,0,0,0],[9E+09,9E+09,9E+09,9E+09,9E+09,9E+09]];
  CONST robtarget Target_4010:=[[891.374984158,312.91563679,660.090342283],[0,0,1,0],[0,0,0,0],[9E+09,9E+09,9E+09,9E+09,9E+09,9E+09]];
  CONST robtarget Target_4020:=[[891.374984158,302.91563679,660.090342283],[0,0,1,0],[0,0,0,0],[9E+09,9E+09,9E+09,9E+09,9E+09,9E+09]];
  CONST robtarget Target_4030:=[[891.374984158,292.91563679,660.090342283],[0,0,1,0],[0,0,0,0],[9E+09,9E+09,9E+09,9E+09,9E+09,9E+09]];
  CONST robtarget Target_4040:=[[891.374984158,282.91563679,660.090342283],[0,0,1,0],[0,0,0,0],[9E+09,9E+09,9E+09,9E+09,9E+09,9E+09]];
  CONST robtarget Target_4050:=[[891.374984158,272.91563679,660.090342283],[0,0,1,0],[0,0,0,0],[9E+09,9E+09,9E+09,9E+09,9E+09,9E+09]];
  CONST robtarget Target_4060:=[[891.374984158,262.91563679,660.090342283],[0,0,1,0],[0,0,0,0],[9E+09,9E+09,9E+09,9E+09,9E+09,9E+09]];
  CONST robtarget Target_4070:=[[891.374984158,252.91563679,660.090342283],[0,0,1,0],[0,0,0,0],[9E+09,9E+09,9E+09,9E+09,9E+09,9E+09]];
  CONST robtarget Target_4080:=[[891.374984158,242.91563679,660.090342283],[0,0,1,0],[0,0,0,0],[9E+09,9E+09,9E+09,9E+09,9E+09,9E+09]];
  CONST robtarget Target_4090:=[[891.374984158,232.91563679,660.090342283],[0,0,1,0],[0,0,0,0],[9E+09,9E+09,9E+09,9E+09,9E+09,9E+09]];
  CONST robtarget Target_4100:=[[891.374984158,222.91563679,660.090342283],[0,0,1,0],[0,0,0,0],[9E+09,9E+09,9E+09,9E+09,9E+09,9E+09]];
  CONST robtarget Target_4110:=[[891.374984158,212.91563679,660.090342283],[0,0,1,0],[0,0,0,0],[9E+09,9E+09,9E+09,9E+09,9E+09,9E+09]];
  CONST robtarget Target_4120:=[[891.374984158,202.91563679,660.090342283],[0,0,1,0],[0,0,0,0],[9E+09,9E+09,9E+09,9E+09,9E+09,9E+09]];
  CONST robtarget Target_4130:=[[891.374984158,192.91563679,660.090342283],[0,0,1,0],[0,0,0,0],[9E+09,9E+09,9E+09,9E+09,9E+09,9E+09]];
  CONST robtarget Target_4140:=[[891.374984158,182.91563679,660.090342283],[0,0,1,0],[0,0,0,0],[9E+09,9E+09,9E+09,9E+09,9E+09,9E+09]];
  CONST robtarget Target_4150:=[[891.374984158,172.91563679,660.090342283],[0,0,1,0],[0,0,0,0],[9E+09,9E+09,9E+09,9E+09,9E+09,9E+09]];
  CONST robtarget Target_4160:=[[891.374984158,162.91563679,660.090342283],[0,0,1,0],[0,0,0,0],[9E+09,9E+09,9E+09,9E+09,9E+09,9E+09]];
  CONST robtarget Target_4170:=[[891.374984158,152.91563679,660.090342283],[0,0,1,0],[0,0,0,0],[9E+09,9E+09,9E+09,9E+09,9E+09,9E+09]];
  CONST robtarget Target_4180:=[[891.374984158,142.91563679,660.090342283],[0,0,1,0],[0,0,0,0],[9E+09,9E+09,9E+09,9E+09,9E+09,9E+09]];
  CONST robtarget Target_4190:=[[891.374984158,132.91563679,660.090342283],[0,0,1,0],[0,0,0,0],[9E+09,9E+09,9E+09,9E+09,9E+09,9E+09]];
  CONST robtarget Target_4200:=[[891.374984158,122.91563679,660.090342283],[0,0,1,0],[0,0,0,0],[9E+09,9E+09,9E+09,9E+09,9E+09,9E+09]];
  CONST robtarget Target_4210:=[[891.374984158,112.91563679,660.090342283],[0,0,1,0],[0,0,0,0],[9E+09,9E+09,9E+09,9E+09,9E+09,9E+09]];
  CONST robtarget Target_4220:=[[891.374984158,102.91563679,660.090342283],[0,0,1,0],[0,0,0,0],[9E+09,9E+09,9E+09,9E+09,9E+09,9E+09]];
  CONST robtarget Target_4230:=[[891.374984158,92.91563679,660.090342283],[0,0,1,0],[0,0,0,0],[9E+09,9E+09,9E+09,9E+09,9E+09,9E+09]];
  CONST robtarget Target_4240:=[[891.374984158,82.91563679,660.090342283],[0,0,1,0],[0,0,0,0],[9E+09,9E+09,9E+09,9E+09,9E+09,9E+09]];
  CONST robtarget Target_4250:=[[891.374984158,72.91563679,660.090342283],[0,0,1,0],[0,0,0,0],[9E+09,9E+09,9E+09,9E+09,9E+09,9E+09]];
  CONST robtarget Target_4260:=[[891.374984158,62.91563679,660.090342283],[0,0,1,0],[0,0,0,0],[9E+09,9E+09,9E+09,9E+09,9E+09,9E+09]];
  CONST robtarget Target_4270:=[[891.374984158,52.91563679,660.090342283],[0,0,1,0],[0,0,0,0],[9E+09,9E+09,9E+09,9E+09,9E+09,9E+09]];
  CONST robtarget Target_4280:=[[891.374984158,42.91563679,660.090342283],[0,0,1,0],[0,0,0,0],[9E+09,9E+09,9E+09,9E+09,9E+09,9E+09]];
  CONST robtarget Target_4290:=[[891.374984158,32.91563679,660.090342283],[0,0,1,0],[0,0,0,0],[9E+09,9E+09,9E+09,9E+09,9E+09,9E+09]];
  CONST robtarget Target_4300:=[[891.374984158,22.91563679,660.090342283],[0,0,1,0],[0,0,0,0],[9E+09,9E+09,9E+09,9E+09,9E+09,9E+09]];
  CONST robtarget Target_4310:=[[891.374984158,12.91563679,660.090342283],[0,0,1,0],[0,0,0,0],[9E+09,9E+09,9E+09,9E+09,9E+09,9E+09]];
  CONST robtarget Target_4320:=[[891.374984158,2.91563679,660.090342283],[0,0,1,0],[0,0,0,0],[9E+09,9E+09,9E+09,9E+09,9E+09,9E+09]];
  CONST robtarget Target_4330:=[[891.374984158,-7.08436321,660.090342283],[0,0,1,0],[0,0,0,0],[9E+09,9E+09,9E+09,9E+09,9E+09,9E+09]];
  CONST robtarget Target_4340:=[[891.374984158,-17.08436321,660.090342283],[0,0,1,0],[0,0,0,0],[9E+09,9E+09,9E+09,9E+09,9E+09,9E+09]];
  CONST robtarget Target_4350:=[[891.374984158,-27.08436321,660.090342283],[0,0,1,0],[0,0,0,0],[9E+09,9E+09,9E+09,9E+09,9E+09,9E+09]];
  CONST robtarget Target_4360:=[[891.374984158,-37.08436321,660.090342283],[0,0,1,0],[0,0,0,0],[9E+09,9E+09,9E+09,9E+09,9E+09,9E+09]];
  CONST robtarget Target_4370:=[[891.374984158,-47.08436321,660.090342283],[0,0,1,0],[0,0,0,0],[9E+09,9E+09,9E+09,9E+09,9E+09,9E+09]];
  CONST robtarget Target_4380:=[[891.374984158,-57.08436321,660.090342283],[0,0,1,0],[0,0,0,0],[9E+09,9E+09,9E+09,9E+09,9E+09,9E+09]];
  CONST robtarget Target_4390:=[[891.374984158,-67.08436321,660.090342283],[0,0,1,0],[0,0,0,0],[9E+09,9E+09,9E+09,9E+09,9E+09,9E+09]];
  CONST robtarget Target_4400:=[[891.374984158,-77.08436321,660.090342283],[0,0,1,0],[0,0,0,0],[9E+09,9E+09,9E+09,9E+09,9E+09,9E+09]];
  CONST robtarget Target_4410:=[[891.374984158,-87.08436321,660.090342283],[0,0,1,0],[0,0,0,0],[9E+09,9E+09,9E+09,9E+09,9E+09,9E+09]];
  CONST robtarget Target_4420:=[[891.374906076,-87.084360951,797.370389046],[0.000000055,-0.000000002,1,-0.000000004],[-1,0,-1,0],[9E+09,9E+09,9E+09,9E+09,9E+09,9E+09]];
  CONST robtarget Target_4430:=[[666.373921465,-87.084344276,797.370380986],[0.000000117,-0.000000009,1,-0.000000004],[-1,0,-1,0],[9E+09,9E+09,9E+09,9E+09,9E+09,9E+09]];
  CONST robtarget Target_4440:=[[505.687734585,-87.084357373,797.370386314],[0.000000157,-0.000000005,1,-0.000000007],[-1,0,-1,0],[9E+09,9E+09,9E+09,9E+09,9E+09,9E+09]];
  CONST robtarget Target_4450:=[[387.54726521,-133.684385852,700.090294402],[0.00000026,-0.000000009,1,-0.000000013],[-1,0,-1,0],[9E+09,9E+09,9E+09,9E+09,9E+09,9E+09]];
  CONST robtarget Target_4460:=[[373.374984158,-133.68436321,660.090342283],[0.00000026,-0.000000009,1,-0.000000013],[0,0,0,0],[9E+09,9E+09,9E+09,9E+09,9E+09,9E+09]];
  CONST robtarget Target_4470:=[[373.374984158,-143.68436321,660.090342283],[0.00000026,-0.000000009,1,-0.000000013],[0,0,0,0],[9E+09,9E+09,9E+09,9E+09,9E+09,9E+09]];
  CONST robtarget Target_4480:=[[373.374984158,-153.68436321,660.090342283],[0.00000026,-0.000000009,1,-0.000000013],[0,0,0,0],[9E+09,9E+09,9E+09,9E+09,9E+09,9E+09]];
  CONST robtarget Target_4490:=[[373.374984158,-163.68436321,660.090342283],[0.00000026,-0.000000009,1,-0.000000013],[0,0,0,0],[9E+09,9E+09,9E+09,9E+09,9E+09,9E+09]];
  CONST robtarget Target_4500:=[[373.374984158,-173.68436321,660.090342283],[0.00000026,-0.000000009,1,-0.000000013],[0,0,0,0],[9E+09,9E+09,9E+09,9E+09,9E+09,9E+09]];
  CONST robtarget Target_4510:=[[373.374984158,-183.68436321,660.090342283],[0.00000026,-0.000000009,1,-0.000000013],[0,0,0,0],[9E+09,9E+09,9E+09,9E+09,9E+09,9E+09]];
  CONST robtarget Target_4520:=[[373.374984158,-193.68436321,660.090342283],[0.00000026,-0.000000009,1,-0.000000013],[0,0,0,0],[9E+09,9E+09,9E+09,9E+09,9E+09,9E+09]];
  CONST robtarget Target_4530:=[[373.374984158,-203.68436321,660.090342283],[0.00000026,-0.000000009,1,-0.000000013],[0,0,0,0],[9E+09,9E+09,9E+09,9E+09,9E+09,9E+09]];
  CONST robtarget Target_4540:=[[373.374984158,-213.68436321,660.090342283],[0.00000026,-0.000000009,1,-0.000000013],[0,0,0,0],[9E+09,9E+09,9E+09,9E+09,9E+09,9E+09]];
  CONST robtarget Target_4550:=[[373.374984158,-223.68436321,660.090342283],[0.00000026,-0.000000009,1,-0.000000013],[0,0,0,0],[9E+09,9E+09,9E+09,9E+09,9E+09,9E+09]];
  CONST robtarget Target_4560:=[[373.374984158,-233.68436321,660.090342283],[0.00000026,-0.000000009,1,-0.000000013],[0,0,0,0],[9E+09,9E+09,9E+09,9E+09,9E+09,9E+09]];
  CONST robtarget Target_4570:=[[373.374984158,-243.68436321,660.090342283],[0.00000026,-0.000000009,1,-0.000000013],[0,0,0,0],[9E+09,9E+09,9E+09,9E+09,9E+09,9E+09]];
  CONST robtarget Target_4580:=[[373.374984158,-253.68436321,660.090342283],[0.00000026,-0.000000009,1,-0.000000013],[0,0,0,0],[9E+09,9E+09,9E+09,9E+09,9E+09,9E+09]];
  CONST robtarget Target_4590:=[[373.374984158,-263.68436321,660.090342283],[0.00000026,-0.000000009,1,-0.000000013],[0,0,0,0],[9E+09,9E+09,9E+09,9E+09,9E+09,9E+09]];
  CONST robtarget Target_4600:=[[373.374984158,-273.68436321,660.090342283],[0.00000026,-0.000000009,1,-0.000000013],[0,0,0,0],[9E+09,9E+09,9E+09,9E+09,9E+09,9E+09]];
  CONST robtarget Target_4610:=[[373.374984158,-283.68436321,660.090342283],[0.00000026,-0.000000009,1,-0.000000013],[0,0,0,0],[9E+09,9E+09,9E+09,9E+09,9E+09,9E+09]];
  CONST robtarget Target_4620:=[[373.374984158,-293.68436321,660.090342283],[0.00000026,-0.000000009,1,-0.000000013],[0,0,0,0],[9E+09,9E+09,9E+09,9E+09,9E+09,9E+09]];
  CONST robtarget Target_4630:=[[373.374984158,-303.68436321,660.090342283],[0.00000026,-0.000000009,1,-0.000000013],[0,0,0,0],[9E+09,9E+09,9E+09,9E+09,9E+09,9E+09]];
  CONST robtarget Target_4640:=[[373.374984158,-313.68436321,660.090342283],[0.00000026,-0.000000009,1,-0.000000013],[0,0,0,0],[9E+09,9E+09,9E+09,9E+09,9E+09,9E+09]];
  CONST robtarget Target_4650:=[[373.374984158,-323.68436321,660.090342283],[0.00000026,-0.000000009,1,-0.000000013],[0,0,0,0],[9E+09,9E+09,9E+09,9E+09,9E+09,9E+09]];
  CONST robtarget Target_4660:=[[373.374984158,-333.68436321,660.090342283],[0.00000026,-0.000000009,1,-0.000000013],[0,0,0,0],[9E+09,9E+09,9E+09,9E+09,9E+09,9E+09]];
  CONST robtarget Target_4670:=[[373.374984158,-343.68436321,660.090342283],[0.00000026,-0.000000009,1,-0.000000013],[0,0,0,0],[9E+09,9E+09,9E+09,9E+09,9E+09,9E+09]];
  CONST robtarget Target_4680:=[[373.374984158,-353.68436321,660.090342283],[0.00000026,-0.000000009,1,-0.000000013],[0,0,0,0],[9E+09,9E+09,9E+09,9E+09,9E+09,9E+09]];
  CONST robtarget Target_4690:=[[373.374984158,-363.68436321,660.090342283],[0.00000026,-0.000000009,1,-0.000000013],[0,0,0,0],[9E+09,9E+09,9E+09,9E+09,9E+09,9E+09]];
  CONST robtarget Target_4700:=[[373.374984158,-373.68436321,660.090342283],[0.00000026,-0.000000009,1,-0.000000013],[0,0,0,0],[9E+09,9E+09,9E+09,9E+09,9E+09,9E+09]];
  CONST robtarget Target_4710:=[[373.374984158,-383.68436321,660.090342283],[0.00000026,-0.000000009,1,-0.000000013],[0,0,0,0],[9E+09,9E+09,9E+09,9E+09,9E+09,9E+09]];
  CONST robtarget Target_4720:=[[373.374984158,-393.68436321,660.090342283],[0.00000026,-0.000000009,1,-0.000000013],[0,0,0,0],[9E+09,9E+09,9E+09,9E+09,9E+09,9E+09]];
  CONST robtarget Target_4730:=[[373.374984158,-403.68436321,660.090342283],[0.00000026,-0.000000009,1,-0.000000013],[0,0,0,0],[9E+09,9E+09,9E+09,9E+09,9E+09,9E+09]];
  CONST robtarget Target_4740:=[[373.374984158,-413.68436321,660.090342283],[0.00000026,-0.000000009,1,-0.000000013],[0,0,0,0],[9E+09,9E+09,9E+09,9E+09,9E+09,9E+09]];
  CONST robtarget Target_4750:=[[373.374984158,-423.68436321,660.090342283],[0.00000026,-0.000000009,1,-0.000000013],[0,0,0,0],[9E+09,9E+09,9E+09,9E+09,9E+09,9E+09]];
  CONST robtarget Target_4760:=[[373.374984158,-433.68436321,660.090342283],[0.00000026,-0.000000009,1,-0.000000013],[0,0,0,0],[9E+09,9E+09,9E+09,9E+09,9E+09,9E+09]];
  CONST robtarget Target_4770:=[[373.374984158,-443.68436321,660.090342283],[0.00000026,-0.000000009,1,-0.000000013],[0,0,0,0],[9E+09,9E+09,9E+09,9E+09,9E+09,9E+09]];
  CONST robtarget Target_4780:=[[373.374984158,-453.68436321,660.090342283],[0.00000026,-0.000000009,1,-0.000000013],[0,0,0,0],[9E+09,9E+09,9E+09,9E+09,9E+09,9E+09]];
  CONST robtarget Target_4790:=[[373.374984158,-463.68436321,660.090342283],[0.00000026,-0.000000009,1,-0.000000013],[0,0,0,0],[9E+09,9E+09,9E+09,9E+09,9E+09,9E+09]];
  CONST robtarget Target_4800:=[[373.374984158,-473.68436321,660.090342283],[0.00000026,-0.000000009,1,-0.000000013],[0,0,0,0],[9E+09,9E+09,9E+09,9E+09,9E+09,9E+09]];
  CONST robtarget Target_4810:=[[373.374984158,-483.68436321,660.090342283],[0.00000026,-0.000000009,1,-0.000000013],[0,0,0,0],[9E+09,9E+09,9E+09,9E+09,9E+09,9E+09]];
  CONST robtarget Target_4820:=[[373.374984158,-493.68436321,660.090342283],[0.00000026,-0.000000009,1,-0.000000013],[0,0,0,0],[9E+09,9E+09,9E+09,9E+09,9E+09,9E+09]];
  CONST robtarget Target_4830:=[[373.374984158,-503.68436321,660.090342283],[0.00000026,-0.000000009,1,-0.000000013],[0,0,0,0],[9E+09,9E+09,9E+09,9E+09,9E+09,9E+09]];
  CONST robtarget Target_4840:=[[373.374984158,-513.68436321,660.090342283],[0.00000026,-0.000000009,1,-0.000000013],[0,0,0,0],[9E+09,9E+09,9E+09,9E+09,9E+09,9E+09]];
  CONST robtarget Target_4850:=[[373.374984158,-523.68436321,660.090342283],[0.00000026,-0.000000009,1,-0.000000013],[0,0,0,0],[9E+09,9E+09,9E+09,9E+09,9E+09,9E+09]];
  CONST robtarget Target_4860:=[[373.374984158,-533.68436321,660.090342283],[0.00000026,-0.000000009,1,-0.000000013],[0,0,0,0],[9E+09,9E+09,9E+09,9E+09,9E+09,9E+09]];
  CONST robtarget Target_4870:=[[373.374984158,-543.68436321,660.090342283],[0.00000026,-0.000000009,1,-0.000000013],[0,0,0,0],[9E+09,9E+09,9E+09,9E+09,9E+09,9E+09]];
  CONST robtarget Target_4880:=[[373.374984158,-553.68436321,660.090342283],[0.00000026,-0.000000009,1,-0.000000013],[0,0,0,0],[9E+09,9E+09,9E+09,9E+09,9E+09,9E+09]];
  CONST robtarget Target_4890:=[[373.374984158,-563.68436321,660.090342283],[0.00000026,-0.000000009,1,-0.000000013],[0,0,0,0],[9E+09,9E+09,9E+09,9E+09,9E+09,9E+09]];
  CONST robtarget Target_4900:=[[373.374984158,-573.68436321,660.090342283],[0.00000026,-0.000000009,1,-0.000000013],[0,0,0,0],[9E+09,9E+09,9E+09,9E+09,9E+09,9E+09]];
  CONST robtarget Home:=[[425.032332,0,1217.172029124],[0.050595114,0,0.998719247,0],[0,0,0,0],[9E+09,9E+09,9E+09,9E+09,9E+09,9E+09]];
  CONST robtarget Target_4910:=[[891.374902342,-133.684394351,765.953436944],[0.00000006,-0.000000005,1,0.000000003],[-1,0,-1,0],[9E+09,9E+09,9E+09,9E+09,9E+09,9E+09]];
  CONST robtarget Target_4920:=[[373.374971985,352.915599084,751.160957312],[0.000000124,-0.000000025,1,0.00000003],[0,-1,0,0],[9E+09,9E+09,9E+09,9E+09,9E+09,9E+09]];
  PROC Path_V1()
    MoveL Target_520,v50,fine,AW_Gun\WObj:=wobj0;
    MoveL Target_510,v50,fine,AW_Gun\WObj:=wobj0;
    MoveL Target_500,v50,fine,AW_Gun\WObj:=wobj0;
    MoveL Target_490,v50,fine,AW_Gun\WObj:=wobj0;
    MoveL Target_480,v50,fine,AW_Gun\WObj:=wobj0;
    MoveL Target_470,v50,fine,AW_Gun\WObj:=wobj0;
    MoveL Target_460,v50,fine,AW_Gun\WObj:=wobj0;
    MoveL Target_450,v50,fine,AW_Gun\WObj:=wobj0;
    MoveL Target_440,v50,fine,AW_Gun\WObj:=wobj0;
    MoveL Target_430,v50,fine,AW_Gun\WObj:=wobj0;
    MoveL Target_420,v50,fine,AW_Gun\WObj:=wobj0;
    MoveL Target_410,v50,fine,AW_Gun\WObj:=wobj0;
    MoveL Target_400,v50,fine,AW_Gun\WObj:=wobj0;
    MoveL Target_390,v50,fine,AW_Gun\WObj:=wobj0;
    MoveL Target_380,v50,fine,AW_Gun\WObj:=wobj0;
    MoveL Target_370,v50,fine,AW_Gun\WObj:=wobj0;
    MoveL Target_360,v50,fine,AW_Gun\WObj:=wobj0;
    MoveL Target_350,v50,fine,AW_Gun\WObj:=wobj0;
    MoveL Target_340,v50,fine,AW_Gun\WObj:=wobj0;
    MoveL Target_330,v50,fine,AW_Gun\WObj:=wobj0;
    MoveL Target_320,v50,fine,AW_Gun\WObj:=wobj0;
    MoveL Target_310,v50,fine,AW_Gun\WObj:=wobj0;
    MoveL Target_300,v50,fine,AW_Gun\WObj:=wobj0;
    MoveL Target_290,v50,fine,AW_Gun\WObj:=wobj0;
    MoveL Target_280,v50,fine,AW_Gun\WObj:=wobj0;
    MoveL Target_270,v50,fine,AW_Gun\WObj:=wobj0;
    MoveL Target_260,v50,fine,AW_Gun\WObj:=wobj0;
    MoveL Target_250,v50,fine,AW_Gun\WObj:=wobj0;
    MoveL Target_240,v50,fine,AW_Gun\WObj:=wobj0;
    MoveL Target_230,v50,fine,AW_Gun\WObj:=wobj0;
    MoveL Target_220,v50,fine,AW_Gun\WObj:=wobj0;
    MoveL Target_210,v50,fine,AW_Gun\WObj:=wobj0;
    MoveL Target_200,v50,fine,AW_Gun\WObj:=wobj0;
    MoveL Target_190,v50,fine,AW_Gun\WObj:=wobj0;
    MoveL Target_180,v50,fine,AW_Gun\WObj:=wobj0;
    MoveL Target_170,v50,fine,AW_Gun\WObj:=wobj0;
    MoveL Target_160,v50,fine,AW_Gun\WObj:=wobj0;
    MoveL Target_150,v50,fine,AW_Gun\WObj:=wobj0;
    MoveL Target_140,v50,fine,AW_Gun\WObj:=wobj0;
    MoveL Target_130,v50,fine,AW_Gun\WObj:=wobj0;
    MoveL Target_120,v50,fine,AW_Gun\WObj:=wobj0;
    MoveL Target_110,v50,fine,AW_Gun\WObj:=wobj0;
    MoveL Target_100,v50,fine,AW_Gun\WObj:=wobj0;
    MoveL Target_90,v50,fine,AW_Gun\WObj:=wobj0;
    MoveL Target_80,v50,fine,AW_Gun\WObj:=wobj0;
    MoveL Target_70,v50,fine,AW_Gun\WObj:=wobj0;
    MoveL Target_60,v50,fine,AW_Gun\WObj:=wobj0;
    MoveL Target_50,v50,fine,AW_Gun\WObj:=wobj0;
    MoveL Target_40,v50,fine,AW_Gun\WObj:=wobj0;
    MoveL Target_30,v50,fine,AW_Gun\WObj:=wobj0;
    MoveL Target_20,v50,fine,AW_Gun\WObj:=wobj0;
    MoveL Target_10,v50,fine,AW_Gun\WObj:=wobj0;
  ENDPROC
  PROC Part_V2()
    MoveL Target_1080,v50,fine,AW_Gun\WObj:=wobj0;
    MoveL Target_1070,v50,fine,AW_Gun\WObj:=wobj0;
    MoveL Target_1060,v50,fine,AW_Gun\WObj:=wobj0;
    MoveL Target_1050,v50,fine,AW_Gun\WObj:=wobj0;
    MoveL Target_1040,v50,fine,AW_Gun\WObj:=wobj0;
    MoveL Target_1030,v50,fine,AW_Gun\WObj:=wobj0;
    MoveL Target_1020,v50,fine,AW_Gun\WObj:=wobj0;
    MoveL Target_1010,v50,fine,AW_Gun\WObj:=wobj0;
    MoveL Target_1000,v50,fine,AW_Gun\WObj:=wobj0;
    MoveL Target_990,v50,fine,AW_Gun\WObj:=wobj0;
    MoveL Target_980,v50,fine,AW_Gun\WObj:=wobj0;
    MoveL Target_970,v50,fine,AW_Gun\WObj:=wobj0;
    MoveL Target_960,v50,fine,AW_Gun\WObj:=wobj0;
    MoveL Target_950,v50,fine,AW_Gun\WObj:=wobj0;
    MoveL Target_940,v50,fine,AW_Gun\WObj:=wobj0;
    MoveL Target_930,v50,fine,AW_Gun\WObj:=wobj0;
    MoveL Target_920,v50,fine,AW_Gun\WObj:=wobj0;
    MoveL Target_910,v50,fine,AW_Gun\WObj:=wobj0;
    MoveL Target_900,v50,fine,AW_Gun\WObj:=wobj0;
    MoveL Target_890,v50,fine,AW_Gun\WObj:=wobj0;
    MoveL Target_880,v50,fine,AW_Gun\WObj:=wobj0;
    MoveL Target_870,v50,fine,AW_Gun\WObj:=wobj0;
    MoveL Target_860,v50,fine,AW_Gun\WObj:=wobj0;
    MoveL Target_850,v50,fine,AW_Gun\WObj:=wobj0;
    MoveL Target_840,v50,fine,AW_Gun\WObj:=wobj0;
    MoveL Target_830,v50,fine,AW_Gun\WObj:=wobj0;
    MoveL Target_820,v50,fine,AW_Gun\WObj:=wobj0;
    MoveL Target_810,v50,fine,AW_Gun\WObj:=wobj0;
    MoveL Target_800,v50,fine,AW_Gun\WObj:=wobj0;
    MoveL Target_790,v50,fine,AW_Gun\WObj:=wobj0;
    MoveL Target_780,v50,fine,AW_Gun\WObj:=wobj0;
    MoveL Target_770,v50,fine,AW_Gun\WObj:=wobj0;
    MoveL Target_760,v50,fine,AW_Gun\WObj:=wobj0;
    MoveL Target_750,v50,fine,AW_Gun\WObj:=wobj0;
    MoveL Target_740,v50,fine,AW_Gun\WObj:=wobj0;
    MoveL Target_730,v50,fine,AW_Gun\WObj:=wobj0;
    MoveL Target_720,v50,fine,AW_Gun\WObj:=wobj0;
    MoveL Target_710,v50,fine,AW_Gun\WObj:=wobj0;
    MoveL Target_700,v50,fine,AW_Gun\WObj:=wobj0;
    MoveL Target_690,v50,fine,AW_Gun\WObj:=wobj0;
    MoveL Target_680,v50,fine,AW_Gun\WObj:=wobj0;
    MoveL Target_670,v50,fine,AW_Gun\WObj:=wobj0;
    MoveL Target_660,v50,fine,AW_Gun\WObj:=wobj0;
    MoveL Target_650,v50,fine,AW_Gun\WObj:=wobj0;
    MoveL Target_640,v50,fine,AW_Gun\WObj:=wobj0;
    MoveL Target_630,v50,fine,AW_Gun\WObj:=wobj0;
    MoveL Target_620,v50,fine,AW_Gun\WObj:=wobj0;
    MoveL Target_610,v50,fine,AW_Gun\WObj:=wobj0;
    MoveL Target_600,v50,fine,AW_Gun\WObj:=wobj0;
    MoveL Target_590,v50,fine,AW_Gun\WObj:=wobj0;
    MoveL Target_580,v50,fine,AW_Gun\WObj:=wobj0;
    MoveL Target_570,v50,fine,AW_Gun\WObj:=wobj0;
  ENDPROC
  PROC Path_V3()
    MoveL Target_1090,v50,fine,AW_Gun\WObj:=wobj0;
    MoveL Target_1100,v50,fine,AW_Gun\WObj:=wobj0;
    MoveL Target_1110,v50,fine,AW_Gun\WObj:=wobj0;
    MoveL Target_1120,v50,fine,AW_Gun\WObj:=wobj0;
    MoveL Target_1130,v50,fine,AW_Gun\WObj:=wobj0;
    MoveL Target_1140,v50,fine,AW_Gun\WObj:=wobj0;
    MoveL Target_1150,v50,fine,AW_Gun\WObj:=wobj0;
    MoveL Target_1160,v50,fine,AW_Gun\WObj:=wobj0;
    MoveL Target_1170,v50,fine,AW_Gun\WObj:=wobj0;
    MoveL Target_1180,v50,fine,AW_Gun\WObj:=wobj0;
    MoveL Target_1190,v50,fine,AW_Gun\WObj:=wobj0;
    MoveL Target_1200,v50,fine,AW_Gun\WObj:=wobj0;
    MoveL Target_1210,v50,fine,AW_Gun\WObj:=wobj0;
    MoveL Target_1220,v50,fine,AW_Gun\WObj:=wobj0;
    MoveL Target_1230,v50,fine,AW_Gun\WObj:=wobj0;
    MoveL Target_1240,v50,fine,AW_Gun\WObj:=wobj0;
    MoveL Target_1250,v50,fine,AW_Gun\WObj:=wobj0;
    MoveL Target_1260,v50,fine,AW_Gun\WObj:=wobj0;
    MoveL Target_1270,v50,fine,AW_Gun\WObj:=wobj0;
    MoveL Target_1280,v50,fine,AW_Gun\WObj:=wobj0;
    MoveL Target_1290,v50,fine,AW_Gun\WObj:=wobj0;
    MoveL Target_1300,v50,fine,AW_Gun\WObj:=wobj0;
    MoveL Target_1310,v50,fine,AW_Gun\WObj:=wobj0;
    MoveL Target_1320,v50,fine,AW_Gun\WObj:=wobj0;
    MoveL Target_1330,v50,fine,AW_Gun\WObj:=wobj0;
    MoveL Target_1340,v50,fine,AW_Gun\WObj:=wobj0;
    MoveL Target_1350,v50,fine,AW_Gun\WObj:=wobj0;
    MoveL Target_1360,v50,fine,AW_Gun\WObj:=wobj0;
    MoveL Target_1370,v50,fine,AW_Gun\WObj:=wobj0;
    MoveL Target_1380,v50,fine,AW_Gun\WObj:=wobj0;
    MoveL Target_1390,v50,fine,AW_Gun\WObj:=wobj0;
    MoveL Target_1400,v50,fine,AW_Gun\WObj:=wobj0;
    MoveL Target_1410,v50,fine,AW_Gun\WObj:=wobj0;
    MoveL Target_1420,v50,fine,AW_Gun\WObj:=wobj0;
    MoveL Target_1430,v50,fine,AW_Gun\WObj:=wobj0;
    MoveL Target_1440,v50,fine,AW_Gun\WObj:=wobj0;
    MoveL Target_1450,v50,fine,AW_Gun\WObj:=wobj0;
    MoveL Target_1460,v50,fine,AW_Gun\WObj:=wobj0;
    MoveL Target_1470,v50,fine,AW_Gun\WObj:=wobj0;
    MoveL Target_1480,v50,fine,AW_Gun\WObj:=wobj0;
    MoveL Target_1490,v50,fine,AW_Gun\WObj:=wobj0;
    MoveL Target_1500,v50,fine,AW_Gun\WObj:=wobj0;
    MoveL Target_1510,v50,fine,AW_Gun\WObj:=wobj0;
    MoveL Target_1520,v50,fine,AW_Gun\WObj:=wobj0;
    MoveL Target_1530,v50,fine,AW_Gun\WObj:=wobj0;
    MoveL Target_1540,v50,fine,AW_Gun\WObj:=wobj0;
    MoveL Target_1550,v50,fine,AW_Gun\WObj:=wobj0;
    MoveL Target_1560,v50,fine,AW_Gun\WObj:=wobj0;
    MoveL Target_1570,v50,fine,AW_Gun\WObj:=wobj0;
    MoveL Target_1580,v50,fine,AW_Gun\WObj:=wobj0;
    MoveL Target_1590,v50,fine,AW_Gun\WObj:=wobj0;
    MoveL Target_1600,v50,fine,AW_Gun\WObj:=wobj0;
  ENDPROC
  PROC Path_V4()
    MoveL Target_2120,v50,fine,AW_Gun\WObj:=wobj0;
    MoveL Target_2110,v20,fine,AW_Gun\WObj:=wobj0;
    MoveL Target_2100,v20,fine,AW_Gun\WObj:=wobj0;
    MoveL Target_2090,v20,fine,AW_Gun\WObj:=wobj0;
    MoveL Target_2080,v20,fine,AW_Gun\WObj:=wobj0;
    MoveL Target_2070,v20,fine,AW_Gun\WObj:=wobj0;
    MoveL Target_2060,v20,fine,AW_Gun\WObj:=wobj0;
    MoveL Target_2050,v20,fine,AW_Gun\WObj:=wobj0;
    MoveL Target_2040,v20,fine,AW_Gun\WObj:=wobj0;
    MoveL Target_2030,v20,fine,AW_Gun\WObj:=wobj0;
    MoveL Target_2020,v20,fine,AW_Gun\WObj:=wobj0;
    MoveL Target_2010,v20,fine,AW_Gun\WObj:=wobj0;
    MoveL Target_2000,v20,fine,AW_Gun\WObj:=wobj0;
    MoveL Target_1990,v20,fine,AW_Gun\WObj:=wobj0;
    MoveL Target_1980,v20,fine,AW_Gun\WObj:=wobj0;
    MoveL Target_1970,v20,fine,AW_Gun\WObj:=wobj0;
    MoveL Target_1960,v20,fine,AW_Gun\WObj:=wobj0;
    MoveL Target_1950,v20,fine,AW_Gun\WObj:=wobj0;
    MoveL Target_1940,v20,fine,AW_Gun\WObj:=wobj0;
    MoveL Target_1930,v20,fine,AW_Gun\WObj:=wobj0;
    MoveL Target_1920,v20,fine,AW_Gun\WObj:=wobj0;
    MoveL Target_1910,v20,fine,AW_Gun\WObj:=wobj0;
    MoveL Target_1900,v20,fine,AW_Gun\WObj:=wobj0;
    MoveL Target_1890,v20,fine,AW_Gun\WObj:=wobj0;
    MoveL Target_1880,v20,fine,AW_Gun\WObj:=wobj0;
    MoveL Target_1870,v20,fine,AW_Gun\WObj:=wobj0;
    MoveL Target_1860,v20,fine,AW_Gun\WObj:=wobj0;
    MoveL Target_1850,v20,fine,AW_Gun\WObj:=wobj0;
    MoveL Target_1840,v20,fine,AW_Gun\WObj:=wobj0;
    MoveL Target_1830,v20,fine,AW_Gun\WObj:=wobj0;
    MoveL Target_1820,v20,fine,AW_Gun\WObj:=wobj0;
    MoveL Target_1810,v20,fine,AW_Gun\WObj:=wobj0;
    MoveL Target_1800,v20,fine,AW_Gun\WObj:=wobj0;
    MoveL Target_1790,v20,fine,AW_Gun\WObj:=wobj0;
    MoveL Target_1780,v20,fine,AW_Gun\WObj:=wobj0;
    MoveL Target_1770,v20,fine,AW_Gun\WObj:=wobj0;
    MoveL Target_1760,v20,fine,AW_Gun\WObj:=wobj0;
    MoveL Target_1750,v20,fine,AW_Gun\WObj:=wobj0;
    MoveL Target_1740,v20,fine,AW_Gun\WObj:=wobj0;
    MoveL Target_1730,v20,fine,AW_Gun\WObj:=wobj0;
    MoveL Target_1720,v20,fine,AW_Gun\WObj:=wobj0;
    MoveL Target_1710,v20,fine,AW_Gun\WObj:=wobj0;
    MoveL Target_1700,v20,fine,AW_Gun\WObj:=wobj0;
    MoveL Target_1690,v20,fine,AW_Gun\WObj:=wobj0;
    MoveL Target_1680,v20,fine,AW_Gun\WObj:=wobj0;
    MoveL Target_1670,v20,fine,AW_Gun\WObj:=wobj0;
    MoveL Target_1660,v20,fine,AW_Gun\WObj:=wobj0;
    MoveL Target_1650,v20,fine,AW_Gun\WObj:=wobj0;
    MoveL Target_1640,v20,fine,AW_Gun\WObj:=wobj0;
    MoveL Target_1630,v20,fine,AW_Gun\WObj:=wobj0;
    MoveL Target_1620,v20,fine,AW_Gun\WObj:=wobj0;
    MoveL Target_1610,v20,fine,AW_Gun\WObj:=wobj0;
  ENDPROC
  PROC Path_HB1()
    MoveL Target_2570,v50,fine,AW_Gun\WObj:=wobj0;
    MoveL Target_2560,v50,fine,AW_Gun\WObj:=wobj0;
    MoveL Target_2550,v50,fine,AW_Gun\WObj:=wobj0;
    MoveL Target_2540,v50,fine,AW_Gun\WObj:=wobj0;
    MoveL Target_2530,v50,fine,AW_Gun\WObj:=wobj0;
    MoveL Target_2520,v50,fine,AW_Gun\WObj:=wobj0;
    MoveL Target_2510,v50,fine,AW_Gun\WObj:=wobj0;
    MoveL Target_2500,v50,fine,AW_Gun\WObj:=wobj0;
    MoveL Target_2490,v50,fine,AW_Gun\WObj:=wobj0;
    MoveL Target_2480,v50,fine,AW_Gun\WObj:=wobj0;
    MoveL Target_2470,v50,fine,AW_Gun\WObj:=wobj0;
    MoveL Target_2460,v50,fine,AW_Gun\WObj:=wobj0;
    MoveL Target_2450,v50,fine,AW_Gun\WObj:=wobj0;
    MoveL Target_2440,v50,fine,AW_Gun\WObj:=wobj0;
    MoveL Target_2430,v50,fine,AW_Gun\WObj:=wobj0;
    MoveL Target_2420,v50,fine,AW_Gun\WObj:=wobj0;
    MoveL Target_2410,v50,fine,AW_Gun\WObj:=wobj0;
    MoveL Target_2400,v50,fine,AW_Gun\WObj:=wobj0;
    MoveL Target_2390,v50,fine,AW_Gun\WObj:=wobj0;
    MoveL Target_2380,v50,fine,AW_Gun\WObj:=wobj0;
    MoveL Target_2370,v50,fine,AW_Gun\WObj:=wobj0;
    MoveL Target_2360,v50,fine,AW_Gun\WObj:=wobj0;
    MoveL Target_2350,v50,fine,AW_Gun\WObj:=wobj0;
    MoveL Target_2340,v50,fine,AW_Gun\WObj:=wobj0;
    MoveL Target_2330,v50,fine,AW_Gun\WObj:=wobj0;
    MoveL Target_2320,v50,fine,AW_Gun\WObj:=wobj0;
    MoveL Target_2310,v50,fine,AW_Gun\WObj:=wobj0;
    MoveL Target_2300,v50,fine,AW_Gun\WObj:=wobj0;
    MoveL Target_2290,v50,fine,AW_Gun\WObj:=wobj0;
    MoveL Target_2280,v50,fine,AW_Gun\WObj:=wobj0;
    MoveL Target_2270,v50,fine,AW_Gun\WObj:=wobj0;
    MoveL Target_2260,v50,fine,AW_Gun\WObj:=wobj0;
    MoveL Target_2250,v50,fine,AW_Gun\WObj:=wobj0;
    MoveL Target_2240,v50,fine,AW_Gun\WObj:=wobj0;
    MoveL Target_2230,v50,fine,AW_Gun\WObj:=wobj0;
    MoveL Target_2220,v50,fine,AW_Gun\WObj:=wobj0;
    MoveL Target_2210,v50,fine,AW_Gun\WObj:=wobj0;
    MoveL Target_2200,v50,fine,AW_Gun\WObj:=wobj0;
    MoveL Target_2190,v50,fine,AW_Gun\WObj:=wobj0;
    MoveL Target_2180,v50,fine,AW_Gun\WObj:=wobj0;
    MoveL Target_2170,v50,fine,AW_Gun\WObj:=wobj0;
    MoveL Target_2160,v50,fine,AW_Gun\WObj:=wobj0;
    MoveL Target_2150,v50,fine,AW_Gun\WObj:=wobj0;
    MoveL Target_2140,v50,fine,AW_Gun\WObj:=wobj0;
    MoveL Target_2130,v50,fine,AW_Gun\WObj:=wobj0;
  ENDPROC
  PROC Path_HU2()
    MoveL Target_3020,v50,fine,AW_Gun\WObj:=wobj0;
    MoveL Target_3010,v50,fine,AW_Gun\WObj:=wobj0;
    MoveL Target_3000,v50,fine,AW_Gun\WObj:=wobj0;
    MoveL Target_2990,v50,fine,AW_Gun\WObj:=wobj0;
    MoveL Target_2980,v50,fine,AW_Gun\WObj:=wobj0;
    MoveL Target_2970,v50,fine,AW_Gun\WObj:=wobj0;
    MoveL Target_2960,v50,fine,AW_Gun\WObj:=wobj0;
    MoveL Target_2950,v50,fine,AW_Gun\WObj:=wobj0;
    MoveL Target_2940,v50,fine,AW_Gun\WObj:=wobj0;
    MoveL Target_2930,v50,fine,AW_Gun\WObj:=wobj0;
    MoveL Target_2920,v50,fine,AW_Gun\WObj:=wobj0;
    MoveL Target_2910,v50,fine,AW_Gun\WObj:=wobj0;
    MoveL Target_2900,v50,fine,AW_Gun\WObj:=wobj0;
    MoveL Target_2890,v50,fine,AW_Gun\WObj:=wobj0;
    MoveL Target_2880,v50,fine,AW_Gun\WObj:=wobj0;
    MoveL Target_2870,v50,fine,AW_Gun\WObj:=wobj0;
    MoveL Target_2860,v50,fine,AW_Gun\WObj:=wobj0;
    MoveL Target_2850,v50,fine,AW_Gun\WObj:=wobj0;
    MoveL Target_2840,v50,fine,AW_Gun\WObj:=wobj0;
    MoveL Target_2830,v50,fine,AW_Gun\WObj:=wobj0;
    MoveL Target_2820,v50,fine,AW_Gun\WObj:=wobj0;
    MoveL Target_2810,v50,fine,AW_Gun\WObj:=wobj0;
    MoveL Target_2800,v50,fine,AW_Gun\WObj:=wobj0;
    MoveL Target_2790,v50,fine,AW_Gun\WObj:=wobj0;
    MoveL Target_2780,v50,fine,AW_Gun\WObj:=wobj0;
    MoveL Target_2770,v50,fine,AW_Gun\WObj:=wobj0;
    MoveL Target_2760,v50,fine,AW_Gun\WObj:=wobj0;
    MoveL Target_2750,v50,fine,AW_Gun\WObj:=wobj0;
    MoveL Target_2740,v50,fine,AW_Gun\WObj:=wobj0;
    MoveL Target_2730,v50,fine,AW_Gun\WObj:=wobj0;
    MoveL Target_2720,v50,fine,AW_Gun\WObj:=wobj0;
    MoveL Target_2710,v50,fine,AW_Gun\WObj:=wobj0;
    MoveL Target_2700,v50,fine,AW_Gun\WObj:=wobj0;
    MoveL Target_2690,v50,fine,AW_Gun\WObj:=wobj0;
    MoveL Target_2680,v50,fine,AW_Gun\WObj:=wobj0;
    MoveL Target_2670,v50,fine,AW_Gun\WObj:=wobj0;
    MoveL Target_2660,v50,fine,AW_Gun\WObj:=wobj0;
    MoveL Target_2650,v50,fine,AW_Gun\WObj:=wobj0;
    MoveL Target_2640,v50,fine,AW_Gun\WObj:=wobj0;
    MoveL Target_2630,v50,fine,AW_Gun\WObj:=wobj0;
    MoveL Target_2620,v50,fine,AW_Gun\WObj:=wobj0;
    MoveL Target_2610,v50,fine,AW_Gun\WObj:=wobj0;
    MoveL Target_2600,v50,fine,AW_Gun\WObj:=wobj0;
    MoveL Target_2590,v50,fine,AW_Gun\WObj:=wobj0;
    MoveL Target_2580,v50,fine,AW_Gun\WObj:=wobj0;
  ENDPROC
  PROC Path_HB3()
    MoveL Target_3470,v50,fine,AW_Gun\WObj:=wobj0;
    MoveL Target_3460,v50,fine,AW_Gun\WObj:=wobj0;
    MoveL Target_3450,v50,fine,AW_Gun\WObj:=wobj0;
    MoveL Target_3440,v50,fine,AW_Gun\WObj:=wobj0;
    MoveL Target_3430,v50,fine,AW_Gun\WObj:=wobj0;
    MoveL Target_3420,v50,fine,AW_Gun\WObj:=wobj0;
    MoveL Target_3410,v50,fine,AW_Gun\WObj:=wobj0;
    MoveL Target_3400,v50,fine,AW_Gun\WObj:=wobj0;
    MoveL Target_3390,v50,fine,AW_Gun\WObj:=wobj0;
    MoveL Target_3380,v50,fine,AW_Gun\WObj:=wobj0;
    MoveL Target_3370,v50,fine,AW_Gun\WObj:=wobj0;
    MoveL Target_3360,v50,fine,AW_Gun\WObj:=wobj0;
    MoveL Target_3350,v50,fine,AW_Gun\WObj:=wobj0;
    MoveL Target_3340,v50,fine,AW_Gun\WObj:=wobj0;
    MoveL Target_3330,v50,fine,AW_Gun\WObj:=wobj0;
    MoveL Target_3320,v50,fine,AW_Gun\WObj:=wobj0;
    MoveL Target_3310,v50,fine,AW_Gun\WObj:=wobj0;
    MoveL Target_3300,v50,fine,AW_Gun\WObj:=wobj0;
    MoveL Target_3290,v50,fine,AW_Gun\WObj:=wobj0;
    MoveL Target_3280,v50,fine,AW_Gun\WObj:=wobj0;
    MoveL Target_3270,v50,fine,AW_Gun\WObj:=wobj0;
    MoveL Target_3260,v50,fine,AW_Gun\WObj:=wobj0;
    MoveL Target_3250,v50,fine,AW_Gun\WObj:=wobj0;
    MoveL Target_3240,v50,fine,AW_Gun\WObj:=wobj0;
    MoveL Target_3230,v50,fine,AW_Gun\WObj:=wobj0;
    MoveL Target_3220,v50,fine,AW_Gun\WObj:=wobj0;
    MoveL Target_3210,v50,fine,AW_Gun\WObj:=wobj0;
    MoveL Target_3200,v50,fine,AW_Gun\WObj:=wobj0;
    MoveL Target_3190,v50,fine,AW_Gun\WObj:=wobj0;
    MoveL Target_3180,v50,fine,AW_Gun\WObj:=wobj0;
    MoveL Target_3170,v50,fine,AW_Gun\WObj:=wobj0;
    MoveL Target_3160,v50,fine,AW_Gun\WObj:=wobj0;
    MoveL Target_3150,v50,fine,AW_Gun\WObj:=wobj0;
    MoveL Target_3140,v50,fine,AW_Gun\WObj:=wobj0;
    MoveL Target_3130,v50,fine,AW_Gun\WObj:=wobj0;
    MoveL Target_3120,v50,fine,AW_Gun\WObj:=wobj0;
    MoveL Target_3110,v50,fine,AW_Gun\WObj:=wobj0;
    MoveL Target_3100,v50,fine,AW_Gun\WObj:=wobj0;
    MoveL Target_3090,v50,fine,AW_Gun\WObj:=wobj0;
    MoveL Target_3080,v50,fine,AW_Gun\WObj:=wobj0;
    MoveL Target_3070,v50,fine,AW_Gun\WObj:=wobj0;
    MoveL Target_3060,v50,fine,AW_Gun\WObj:=wobj0;
    MoveL Target_3050,v50,fine,AW_Gun\WObj:=wobj0;
    MoveL Target_3040,v50,fine,AW_Gun\WObj:=wobj0;
    MoveL Target_3030,v50,fine,AW_Gun\WObj:=wobj0;
  ENDPROC
  PROC Path_HU3()
    MoveL Target_3480,v50,fine,AW_Gun\WObj:=wobj0;
    MoveL Target_3490,v50,fine,AW_Gun\WObj:=wobj0;
    MoveL Target_3500,v50,fine,AW_Gun\WObj:=wobj0;
    MoveL Target_3510,v50,fine,AW_Gun\WObj:=wobj0;
    MoveL Target_3520,v50,fine,AW_Gun\WObj:=wobj0;
    MoveL Target_3530,v50,fine,AW_Gun\WObj:=wobj0;
    MoveL Target_3540,v50,fine,AW_Gun\WObj:=wobj0;
    MoveL Target_3550,v50,fine,AW_Gun\WObj:=wobj0;
    MoveL Target_3560,v50,fine,AW_Gun\WObj:=wobj0;
    MoveL Target_3570,v50,fine,AW_Gun\WObj:=wobj0;
    MoveL Target_3580,v50,fine,AW_Gun\WObj:=wobj0;
    MoveL Target_3590,v50,fine,AW_Gun\WObj:=wobj0;
    MoveL Target_3600,v50,fine,AW_Gun\WObj:=wobj0;
    MoveL Target_3610,v50,fine,AW_Gun\WObj:=wobj0;
    MoveL Target_3620,v50,fine,AW_Gun\WObj:=wobj0;
    MoveL Target_3630,v50,fine,AW_Gun\WObj:=wobj0;
    MoveL Target_3640,v50,fine,AW_Gun\WObj:=wobj0;
    MoveL Target_3650,v50,fine,AW_Gun\WObj:=wobj0;
    MoveL Target_3660,v50,fine,AW_Gun\WObj:=wobj0;
    MoveL Target_3670,v50,fine,AW_Gun\WObj:=wobj0;
    MoveL Target_3680,v50,fine,AW_Gun\WObj:=wobj0;
    MoveL Target_3690,v50,fine,AW_Gun\WObj:=wobj0;
    MoveL Target_3700,v50,fine,AW_Gun\WObj:=wobj0;
    MoveL Target_3710,v50,fine,AW_Gun\WObj:=wobj0;
    MoveL Target_3720,v50,fine,AW_Gun\WObj:=wobj0;
    MoveL Target_3730,v50,fine,AW_Gun\WObj:=wobj0;
    MoveL Target_3740,v50,fine,AW_Gun\WObj:=wobj0;
    MoveL Target_3750,v50,fine,AW_Gun\WObj:=wobj0;
    MoveL Target_3760,v50,fine,AW_Gun\WObj:=wobj0;
    MoveL Target_3770,v50,fine,AW_Gun\WObj:=wobj0;
    MoveL Target_3780,v50,fine,AW_Gun\WObj:=wobj0;
    MoveL Target_3790,v50,fine,AW_Gun\WObj:=wobj0;
    MoveL Target_3800,v50,fine,AW_Gun\WObj:=wobj0;
    MoveL Target_3810,v50,fine,AW_Gun\WObj:=wobj0;
    MoveL Target_3820,v50,fine,AW_Gun\WObj:=wobj0;
    MoveL Target_3830,v50,fine,AW_Gun\WObj:=wobj0;
    MoveL Target_3840,v50,fine,AW_Gun\WObj:=wobj0;
    MoveL Target_3850,v50,fine,AW_Gun\WObj:=wobj0;
    MoveL Target_3860,v50,fine,AW_Gun\WObj:=wobj0;
    MoveL Target_3870,v50,fine,AW_Gun\WObj:=wobj0;
    MoveL Target_3880,v50,fine,AW_Gun\WObj:=wobj0;
    MoveL Target_3890,v50,fine,AW_Gun\WObj:=wobj0;
    MoveL Target_3900,v50,fine,AW_Gun\WObj:=wobj0;
    MoveL Target_3910,v50,fine,AW_Gun\WObj:=wobj0;
    MoveL Target_3920,v50,fine,AW_Gun\WObj:=wobj0;
  ENDPROC
  PROC Main()
    From_Home;
    Path_V1;
    Path_HB1;
    Path_Jump1;
    Part_V2;
    Path_HU2;
    Path_Jump2;
    Path_V3;
    Path_HB3;
    Path_V4;
    Path_HU3;
    Path_Rapid1;
    Path_HB2;
    Path_Rapid2;
    Path_HU1;
    To_Home;
  ENDPROC
  PROC Path_Rapid1()
    MoveL Target_3930,v1000,z100,AW_Gun\WObj:=wobj0;
    MoveL Target_3940,v1000,z100,AW_Gun\WObj:=wobj0;
    MoveL Target_3950,v1000,z100,AW_Gun\WObj:=wobj0;
    MoveL Target_3960,v1000,z100,AW_Gun\WObj:=wobj0;
  ENDPROC
  PROC Path_HB2()
    MoveL Target_3970,v50,fine,AW_Gun\WObj:=wobj0;
    MoveL Target_3980,v50,fine,AW_Gun\WObj:=wobj0;
    MoveL Target_3990,v50,fine,AW_Gun\WObj:=wobj0;
    MoveL Target_4000,v50,fine,AW_Gun\WObj:=wobj0;
    MoveL Target_4010,v50,fine,AW_Gun\WObj:=wobj0;
    MoveL Target_4020,v50,fine,AW_Gun\WObj:=wobj0;
    MoveL Target_4030,v50,fine,AW_Gun\WObj:=wobj0;
    MoveL Target_4040,v50,fine,AW_Gun\WObj:=wobj0;
    MoveL Target_4050,v50,fine,AW_Gun\WObj:=wobj0;
    MoveL Target_4060,v50,fine,AW_Gun\WObj:=wobj0;
    MoveL Target_4070,v50,fine,AW_Gun\WObj:=wobj0;
    MoveL Target_4080,v50,fine,AW_Gun\WObj:=wobj0;
    MoveL Target_4090,v50,fine,AW_Gun\WObj:=wobj0;
    MoveL Target_4100,v50,fine,AW_Gun\WObj:=wobj0;
    MoveL Target_4110,v50,fine,AW_Gun\WObj:=wobj0;
    MoveL Target_4120,v50,fine,AW_Gun\WObj:=wobj0;
    MoveL Target_4130,v50,fine,AW_Gun\WObj:=wobj0;
    MoveL Target_4140,v50,fine,AW_Gun\WObj:=wobj0;
    MoveL Target_4150,v50,fine,AW_Gun\WObj:=wobj0;
    MoveL Target_4160,v50,fine,AW_Gun\WObj:=wobj0;
    MoveL Target_4170,v50,fine,AW_Gun\WObj:=wobj0;
    MoveL Target_4180,v50,fine,AW_Gun\WObj:=wobj0;
    MoveL Target_4190,v50,fine,AW_Gun\WObj:=wobj0;
    MoveL Target_4200,v50,fine,AW_Gun\WObj:=wobj0;
    MoveL Target_4210,v50,fine,AW_Gun\WObj:=wobj0;
    MoveL Target_4220,v50,fine,AW_Gun\WObj:=wobj0;
    MoveL Target_4230,v50,fine,AW_Gun\WObj:=wobj0;
    MoveL Target_4240,v50,fine,AW_Gun\WObj:=wobj0;
    MoveL Target_4250,v50,fine,AW_Gun\WObj:=wobj0;
    MoveL Target_4260,v50,fine,AW_Gun\WObj:=wobj0;
    MoveL Target_4270,v50,fine,AW_Gun\WObj:=wobj0;
    MoveL Target_4280,v50,fine,AW_Gun\WObj:=wobj0;
    MoveL Target_4290,v50,fine,AW_Gun\WObj:=wobj0;
    MoveL Target_4300,v50,fine,AW_Gun\WObj:=wobj0;
    MoveL Target_4310,v50,fine,AW_Gun\WObj:=wobj0;
    MoveL Target_4320,v50,fine,AW_Gun\WObj:=wobj0;
    MoveL Target_4330,v50,fine,AW_Gun\WObj:=wobj0;
    MoveL Target_4340,v50,fine,AW_Gun\WObj:=wobj0;
    MoveL Target_4350,v50,fine,AW_Gun\WObj:=wobj0;
    MoveL Target_4360,v50,fine,AW_Gun\WObj:=wobj0;
    MoveL Target_4370,v50,fine,AW_Gun\WObj:=wobj0;
    MoveL Target_4380,v50,fine,AW_Gun\WObj:=wobj0;
    MoveL Target_4390,v50,fine,AW_Gun\WObj:=wobj0;
    MoveL Target_4400,v50,fine,AW_Gun\WObj:=wobj0;
    MoveL Target_4410,v50,fine,AW_Gun\WObj:=wobj0;
  ENDPROC
  PROC Path_Rapid2()
    MoveL Target_4420,v1000,z100,AW_Gun\WObj:=wobj0;
    MoveL Target_4430,v1000,z100,AW_Gun\WObj:=wobj0;
    MoveL Target_4440,v1000,z100,AW_Gun\WObj:=wobj0;
    MoveL Target_4450,v1000,z100,AW_Gun\WObj:=wobj0;
  ENDPROC
  PROC Path_HU1()
    MoveL Target_4460,v50,fine,AW_Gun\WObj:=wobj0;
    MoveL Target_4470,v50,fine,AW_Gun\WObj:=wobj0;
    MoveL Target_4480,v50,fine,AW_Gun\WObj:=wobj0;
    MoveL Target_4490,v50,fine,AW_Gun\WObj:=wobj0;
    MoveL Target_4500,v50,fine,AW_Gun\WObj:=wobj0;
    MoveL Target_4510,v50,fine,AW_Gun\WObj:=wobj0;
    MoveL Target_4520,v50,fine,AW_Gun\WObj:=wobj0;
    MoveL Target_4530,v50,fine,AW_Gun\WObj:=wobj0;
    MoveL Target_4540,v50,fine,AW_Gun\WObj:=wobj0;
    MoveL Target_4550,v50,fine,AW_Gun\WObj:=wobj0;
    MoveL Target_4560,v50,fine,AW_Gun\WObj:=wobj0;
    MoveL Target_4570,v50,fine,AW_Gun\WObj:=wobj0;
    MoveL Target_4580,v50,fine,AW_Gun\WObj:=wobj0;
    MoveL Target_4590,v50,fine,AW_Gun\WObj:=wobj0;
    MoveL Target_4600,v50,fine,AW_Gun\WObj:=wobj0;
    MoveL Target_4610,v50,fine,AW_Gun\WObj:=wobj0;
    MoveL Target_4620,v50,fine,AW_Gun\WObj:=wobj0;
    MoveL Target_4630,v50,fine,AW_Gun\WObj:=wobj0;
    MoveL Target_4640,v50,fine,AW_Gun\WObj:=wobj0;
    MoveL Target_4650,v50,fine,AW_Gun\WObj:=wobj0;
    MoveL Target_4660,v50,fine,AW_Gun\WObj:=wobj0;
    MoveL Target_4670,v50,fine,AW_Gun\WObj:=wobj0;
    MoveL Target_4680,v50,fine,AW_Gun\WObj:=wobj0;
    MoveL Target_4690,v50,fine,AW_Gun\WObj:=wobj0;
    MoveL Target_4700,v50,fine,AW_Gun\WObj:=wobj0;
    MoveL Target_4710,v50,fine,AW_Gun\WObj:=wobj0;
    MoveL Target_4720,v50,fine,AW_Gun\WObj:=wobj0;
    MoveL Target_4730,v50,fine,AW_Gun\WObj:=wobj0;
    MoveL Target_4740,v50,fine,AW_Gun\WObj:=wobj0;
    MoveL Target_4750,v50,fine,AW_Gun\WObj:=wobj0;
    MoveL Target_4760,v50,fine,AW_Gun\WObj:=wobj0;
    MoveL Target_4770,v50,fine,AW_Gun\WObj:=wobj0;
    MoveL Target_4780,v50,fine,AW_Gun\WObj:=wobj0;
    MoveL Target_4790,v50,fine,AW_Gun\WObj:=wobj0;
    MoveL Target_4800,v50,fine,AW_Gun\WObj:=wobj0;
    MoveL Target_4810,v50,fine,AW_Gun\WObj:=wobj0;
    MoveL Target_4820,v50,fine,AW_Gun\WObj:=wobj0;
    MoveL Target_4830,v50,fine,AW_Gun\WObj:=wobj0;
    MoveL Target_4840,v50,fine,AW_Gun\WObj:=wobj0;
    MoveL Target_4850,v50,fine,AW_Gun\WObj:=wobj0;
    MoveL Target_4860,v50,fine,AW_Gun\WObj:=wobj0;
    MoveL Target_4870,v50,fine,AW_Gun\WObj:=wobj0;
    MoveL Target_4880,v50,fine,AW_Gun\WObj:=wobj0;
    MoveL Target_4890,v50,fine,AW_Gun\WObj:=wobj0;
    MoveL Target_4900,v50,fine,AW_Gun\WObj:=wobj0;
  ENDPROC
  PROC From_Home()
    MoveL Home,v1000,z100,AW_Gun\WObj:=wobj0;
    MoveL Target_520,v1000,z100,AW_Gun\WObj:=wobj0;
  ENDPROC
  PROC To_Home()
    MoveL Target_520,v1000,z100,AW_Gun\WObj:=wobj0;
    MoveL Home,v1000,z100,AW_Gun\WObj:=wobj0;
  ENDPROC
  PROC Path_Jump1()
    MoveL Target_4910,v1000,z100,AW_Gun\WObj:=wobj0;
    MoveL Target_1080,v1000,z100,AW_Gun\WObj:=wobj0;
  ENDPROC
  PROC Path_Jump2()
    MoveL Target_4920,v1000,z100,AW_Gun\WObj:=wobj0;
    MoveL Target_1090,v1000,z100,AW_Gun\WObj:=wobj0;
  ENDPROC
ENDMODULE

